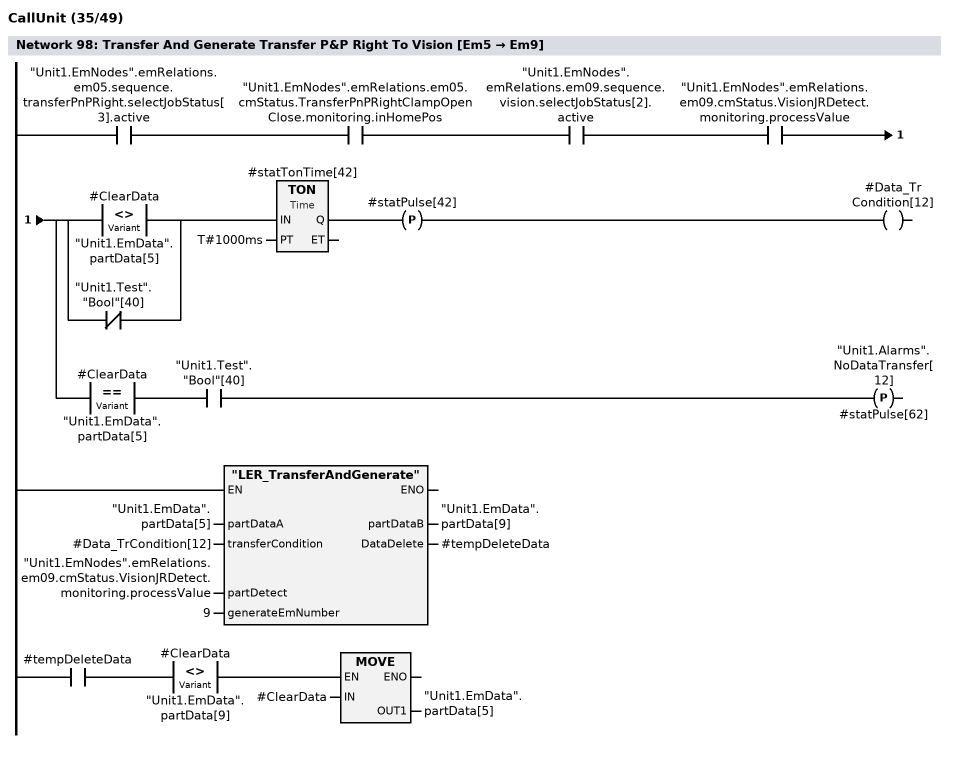
   #_w1 := "Unit1.EmNodes".emRelations.em05.sequence.transferPnPRight.selectJobStatus[3].active AND "Unit1.EmNodes".emRelations.em05.cmStatus.TransferPnPRightClampOpenClose.monitoring.inHomePos AND "Unit1.EmNodes".emRelations.em09.sequence.vision.selectJobStatus[2].active AND "Unit1.EmNodes".emRelations.em09.cmStatus.VisionJRDetect.monitoring.processValue;
   #statTonTime[42].TON(IN := #_w1 AND ((#ClearData <> "Unit1.EmData".partData[5]) OR NOT "Unit1.Test"."Bool"[40]),
                        PT := T#1000ms);
   #_w2 := #statTonTime[42].Q AND NOT #statPulse[42];   // rising edge
   #statPulse[42] := #statTonTime[42].Q;
   #Data_TrCondition[12] := #_w2;
   #_w3 := #_w1 AND (#ClearData = "Unit1.EmData".partData[5]) AND "Unit1.Test"."Bool"[40];
   "Unit1.Alarms".NoDataTransfer[12] := #_w3 AND NOT #statPulse[62];   // rising edge
   #statPulse[62] := #_w3;
   "LER_TransferAndGenerate"(partDataA := "Unit1.EmData".partData[5],
                           transferCondition := #Data_TrCondition[12],
                           partDetect := "Unit1.EmNodes".emRelations.em09.cmStatus.VisionJRDetect.monitoring.processValue,
                           generateEmNumber := 9,
                           partDataB => "Unit1.EmData".partData[9],
                           DataDelete => #tempDeleteData);
   IF #tempDeleteData AND (#ClearData <> "Unit1.EmData".partData[9]) THEN
       "Unit1.EmData".partData[5] := #ClearData;
   END_IF;
END_REGION

REGION Network 99: Transfer And Generate Vision To Transfer P&P Right [Em9 → Em5]
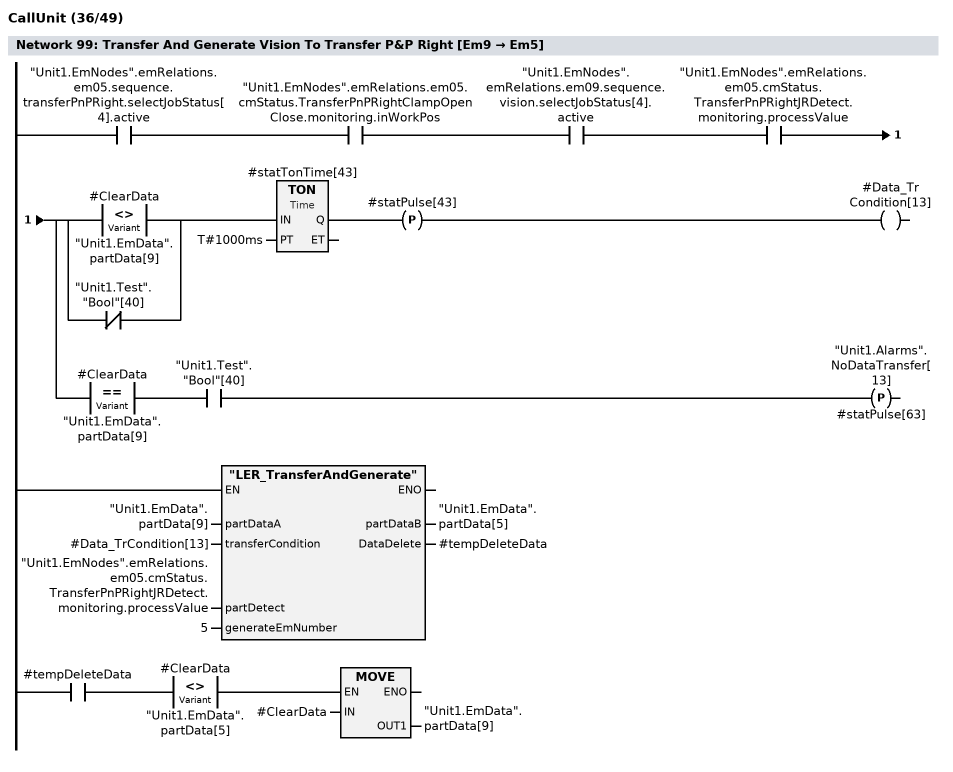
   #_w1 := "Unit1.EmNodes".emRelations.em05.sequence.transferPnPRight.selectJobStatus[4].active AND "Unit1.EmNodes".emRelations.em05.cmStatus.TransferPnPRightClampOpenClose.monitoring.inWorkPos AND "Unit1.EmNodes".emRelations.em09.sequence.vision.selectJobStatus[4].active AND "Unit1.EmNodes".emRelations.em05.cmStatus.TransferPnPRightJRDetect.monitoring.processValue;
   #statTonTime[43].TON(IN := #_w1 AND ((#ClearData <> "Unit1.EmData".partData[9]) OR NOT "Unit1.Test"."Bool"[40]),
                        PT := T#1000ms);
   #_w2 := #statTonTime[43].Q AND NOT #statPulse[43];   // rising edge
   #statPulse[43] := #statTonTime[43].Q;
   #Data_TrCondition[13] := #_w2;
   #_w3 := #_w1 AND (#ClearData = "Unit1.EmData".partData[9]) AND "Unit1.Test"."Bool"[40];
   "Unit1.Alarms".NoDataTransfer[13] := #_w3 AND NOT #statPulse[63];   // rising edge
   #statPulse[63] := #_w3;
   "LER_TransferAndGenerate"(partDataA := "Unit1.EmData".partData[9],
                           transferCondition := #Data_TrCondition[13],
                           partDetect := "Unit1.EmNodes".emRelations.em05.cmStatus.TransferPnPRightJRDetect.monitoring.processValue,
                           generateEmNumber := 5,
                           partDataB => "Unit1.EmData".partData[5],
                           DataDelete => #tempDeleteData);
   IF #tempDeleteData AND (#ClearData <> "Unit1.EmData".partData[5]) THEN
       "Unit1.EmData".partData[9] := #ClearData;
   END_IF;
END_REGION

REGION Network 100: Transfer And Generate Transfer P&P Right To Laser Mark [Em5 → Em10]
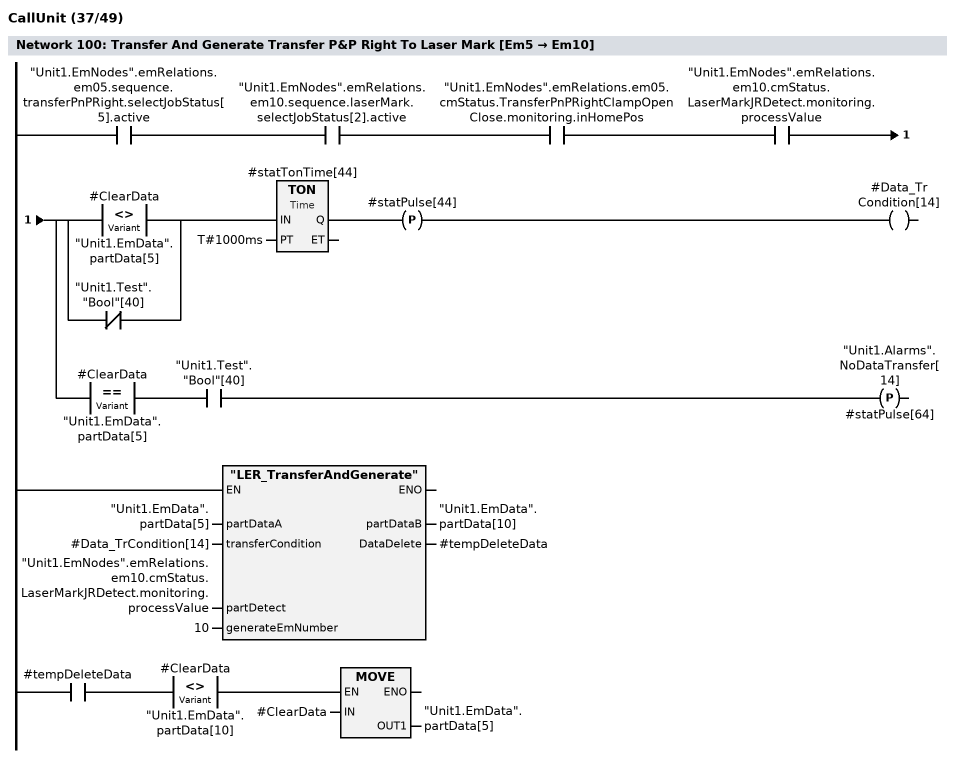
   #_w1 := "Unit1.EmNodes".emRelations.em05.sequence.transferPnPRight.selectJobStatus[5].active AND "Unit1.EmNodes".emRelations.em10.sequence.laserMark.selectJobStatus[2].active AND "Unit1.EmNodes".emRelations.em05.cmStatus.TransferPnPRightClampOpenClose.monitoring.inHomePos AND "Unit1.EmNodes".emRelations.em10.cmStatus.LaserMarkJRDetect.monitoring.processValue;
   #statTonTime[44].TON(IN := #_w1 AND ((#ClearData <> "Unit1.EmData".partData[5]) OR NOT "Unit1.Test"."Bool"[40]),
                        PT := T#1000ms);
   #_w2 := #statTonTime[44].Q AND NOT #statPulse[44];   // rising edge
   #statPulse[44] := #statTonTime[44].Q;
   #Data_TrCondition[14] := #_w2;
   #_w3 := #_w1 AND (#ClearData = "Unit1.EmData".partData[5]) AND "Unit1.Test"."Bool"[40];
   "Unit1.Alarms".NoDataTransfer[14] := #_w3 AND NOT #statPulse[64];   // rising edge
   #statPulse[64] := #_w3;
   "LER_TransferAndGenerate"(partDataA := "Unit1.EmData".partData[5],
                           transferCondition := #Data_TrCondition[14],
                           partDetect := "Unit1.EmNodes".emRelations.em10.cmStatus.LaserMarkJRDetect.monitoring.processValue,
                           generateEmNumber := 10,
                           partDataB => "Unit1.EmData".partData[10],
                           DataDelete => #tempDeleteData);
   IF #tempDeleteData AND (#ClearData <> "Unit1.EmData".partData[10]) THEN
       "Unit1.EmData".partData[5] := #ClearData;
   END_IF;
END_REGION

REGION Network 101: Transfer And Generate Laser Mark To Transfer P&P Right [Em10 → Em5]
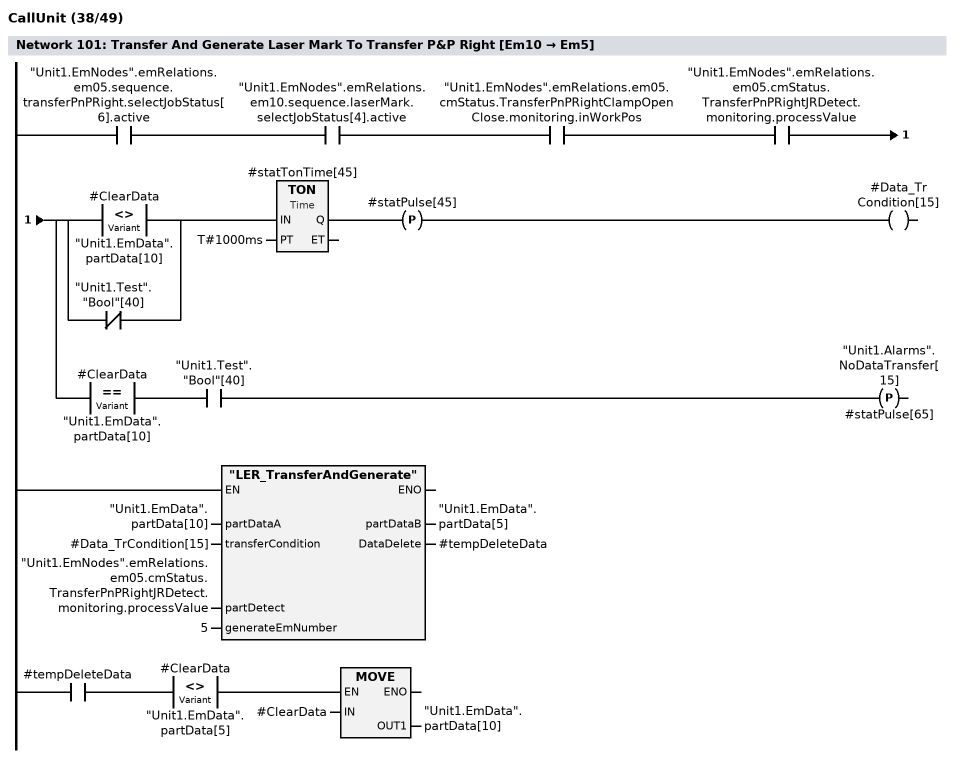
   #_w1 := "Unit1.EmNodes".emRelations.em05.sequence.transferPnPRight.selectJobStatus[6].active AND "Unit1.EmNodes".emRelations.em10.sequence.laserMark.selectJobStatus[4].active AND "Unit1.EmNodes".emRelations.em05.cmStatus.TransferPnPRightClampOpenClose.monitoring.inWorkPos AND "Unit1.EmNodes".emRelations.em05.cmStatus.TransferPnPRightJRDetect.monitoring.processValue;
   #statTonTime[45].TON(IN := #_w1 AND ((#ClearData <> "Unit1.EmData".partData[10]) OR NOT "Unit1.Test"."Bool"[40]),
                        PT := T#1000ms);
   #_w2 := #statTonTime[45].Q AND NOT #statPulse[45];   // rising edge
   #statPulse[45] := #statTonTime[45].Q;
   #Data_TrCondition[15] := #_w2;
   #_w3 := #_w1 AND (#ClearData = "Unit1.EmData".partData[10]) AND "Unit1.Test"."Bool"[40];
   "Unit1.Alarms".NoDataTransfer[15] := #_w3 AND NOT #statPulse[65];   // rising edge
   #statPulse[65] := #_w3;
   "LER_TransferAndGenerate"(partDataA := "Unit1.EmData".partData[10],
                           transferCondition := #Data_TrCondition[15],
                           partDetect := "Unit1.EmNodes".emRelations.em05.cmStatus.TransferPnPRightJRDetect.monitoring.processValue,
                           generateEmNumber := 5,
                           partDataB => "Unit1.EmData".partData[5],
                           DataDelete => #tempDeleteData);
   IF #tempDeleteData AND (#ClearData <> "Unit1.EmData".partData[5]) THEN
       "Unit1.EmData".partData[10] := #ClearData;
   END_IF;
END_REGION

REGION Network 102: Transfer And Generate Transfer P&P Right To Weight Check [Em5 → Em11]
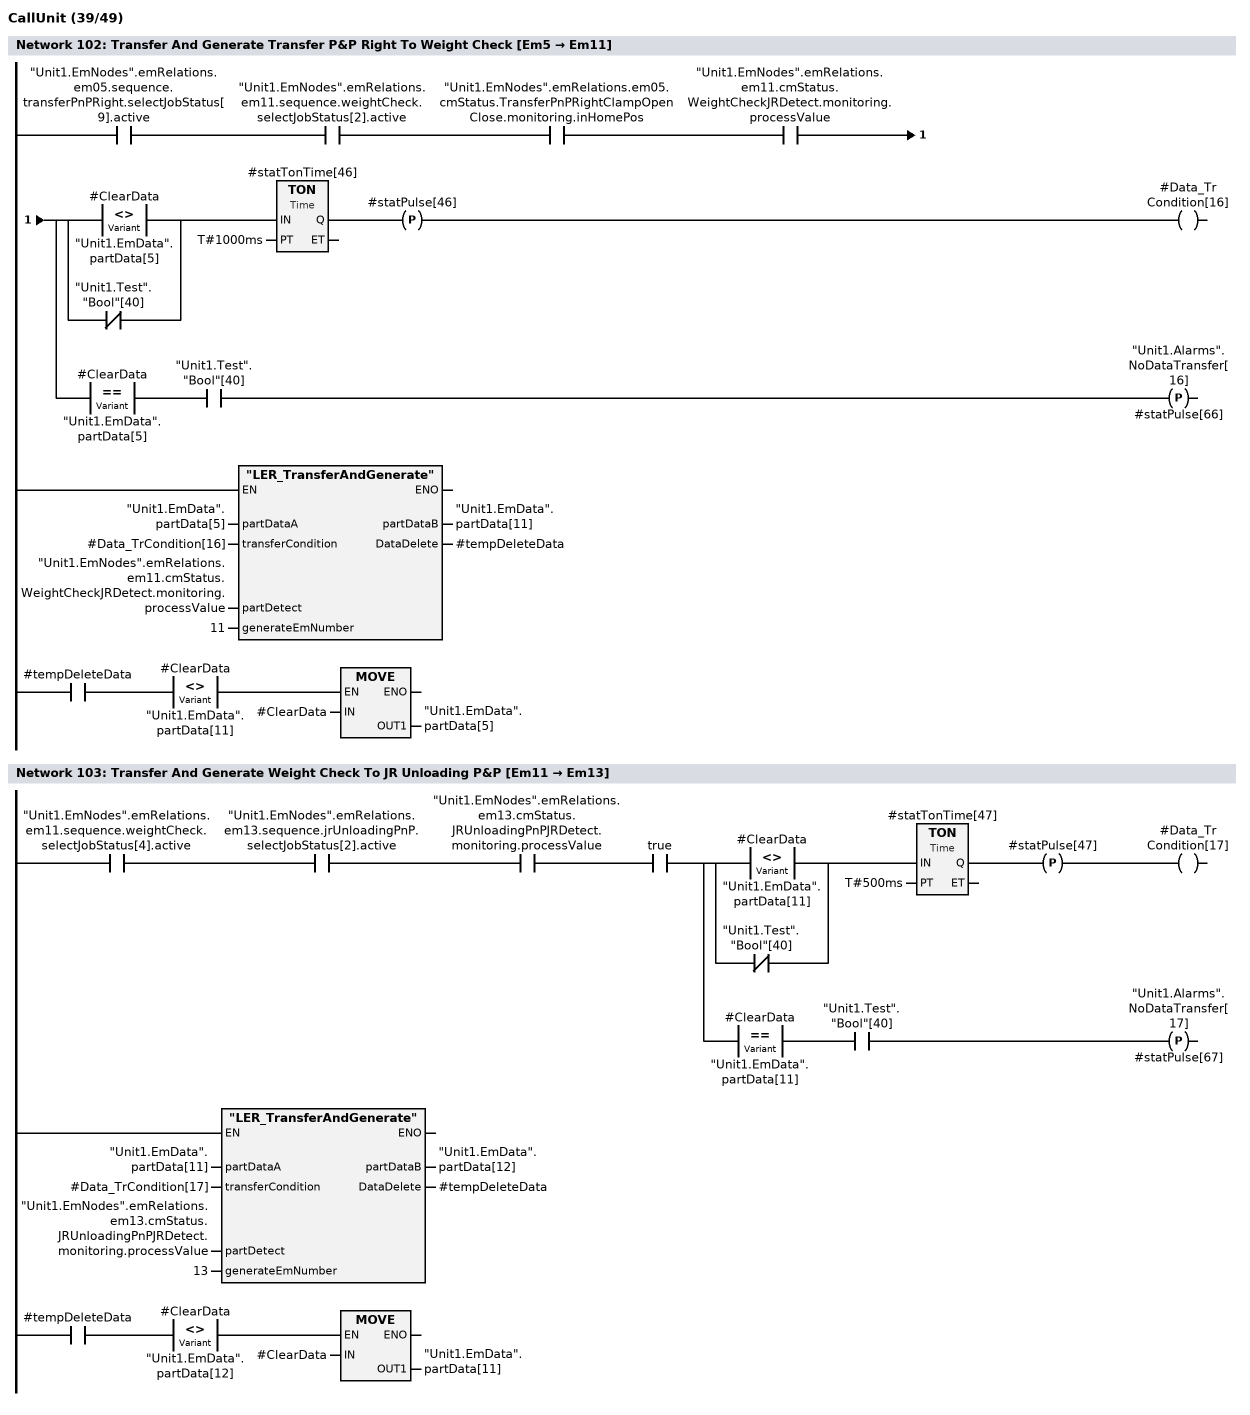
   #_w1 := "Unit1.EmNodes".emRelations.em05.sequence.transferPnPRight.selectJobStatus[9].active AND "Unit1.EmNodes".emRelations.em11.sequence.weightCheck.selectJobStatus[2].active AND "Unit1.EmNodes".emRelations.em05.cmStatus.TransferPnPRightClampOpenClose.monitoring.inHomePos AND "Unit1.EmNodes".emRelations.em11.cmStatus.WeightCheckJRDetect.monitoring.processValue;
   #statTonTime[46].TON(IN := #_w1 AND ((#ClearData <> "Unit1.EmData".partData[5]) OR NOT "Unit1.Test"."Bool"[40]),
                        PT := T#1000ms);
   #_w2 := #statTonTime[46].Q AND NOT #statPulse[46];   // rising edge
   #statPulse[46] := #statTonTime[46].Q;
   #Data_TrCondition[16] := #_w2;
   #_w3 := #_w1 AND (#ClearData = "Unit1.EmData".partData[5]) AND "Unit1.Test"."Bool"[40];
   "Unit1.Alarms".NoDataTransfer[16] := #_w3 AND NOT #statPulse[66];   // rising edge
   #statPulse[66] := #_w3;
   "LER_TransferAndGenerate"(partDataA := "Unit1.EmData".partData[5],
                           transferCondition := #Data_TrCondition[16],
                           partDetect := "Unit1.EmNodes".emRelations.em11.cmStatus.WeightCheckJRDetect.monitoring.processValue,
                           generateEmNumber := 11,
                           partDataB => "Unit1.EmData".partData[11],
                           DataDelete => #tempDeleteData);
   IF #tempDeleteData AND (#ClearData <> "Unit1.EmData".partData[11]) THEN
       "Unit1.EmData".partData[5] := #ClearData;
   END_IF;
END_REGION

REGION Network 103: Transfer And Generate Weight Check To JR Unloading P&P [Em11 → Em13]
   #_w1 := "Unit1.EmNodes".emRelations.em11.sequence.weightCheck.selectJobStatus[4].active AND "Unit1.EmNodes".emRelations.em13.sequence.jrUnloadingPnP.selectJobStatus[2].active AND "Unit1.EmNodes".emRelations.em13.cmStatus.JRUnloadingPnPJRDetect.monitoring.processValue AND true;
   #statTonTime[47].TON(IN := #_w1 AND ((#ClearData <> "Unit1.EmData".partData[11]) OR NOT "Unit1.Test"."Bool"[40]),
                        PT := T#500ms);
   #_w2 := #statTonTime[47].Q AND NOT #statPulse[47];   // rising edge
   #statPulse[47] := #statTonTime[47].Q;
   #Data_TrCondition[17] := #_w2;
   #_w3 := #_w1 AND (#ClearData = "Unit1.EmData".partData[11]) AND "Unit1.Test"."Bool"[40];
   "Unit1.Alarms".NoDataTransfer[17] := #_w3 AND NOT #statPulse[67];   // rising edge
   #statPulse[67] := #_w3;
   "LER_TransferAndGenerate"(partDataA := "Unit1.EmData".partData[11],
                           transferCondition := #Data_TrCondition[17],
                           partDetect := "Unit1.EmNodes".emRelations.em13.cmStatus.JRUnloadingPnPJRDetect.monitoring.processValue,
                           generateEmNumber := 13,
                           partDataB => "Unit1.EmData".partData[12],
                           DataDelete => #tempDeleteData);
   IF #tempDeleteData AND (#ClearData <> "Unit1.EmData".partData[12]) THEN
       "Unit1.EmData".partData[11] := #ClearData;
   END_IF;
END_REGION

REGION Network 104: Transfer And Generate JR Unloading P&P To ConveyorA [Em13 → ConveyorA]
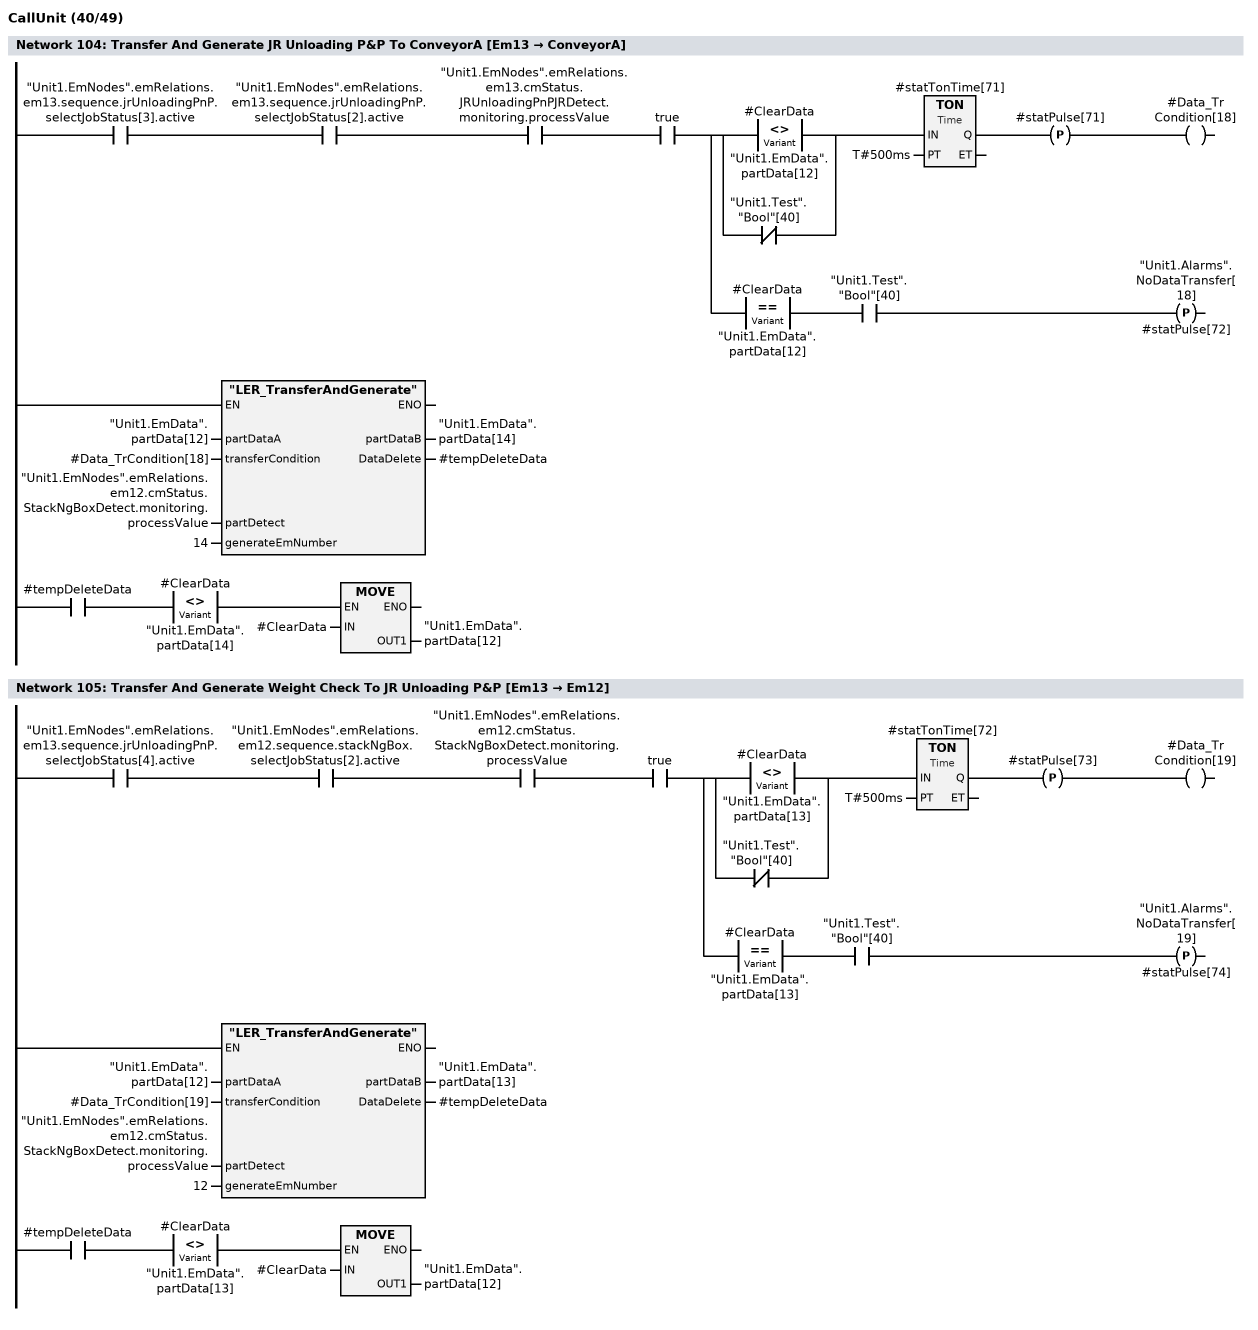
   #_w1 := "Unit1.EmNodes".emRelations.em13.sequence.jrUnloadingPnP.selectJobStatus[3].active AND "Unit1.EmNodes".emRelations.em13.sequence.jrUnloadingPnP.selectJobStatus[2].active AND "Unit1.EmNodes".emRelations.em13.cmStatus.JRUnloadingPnPJRDetect.monitoring.processValue AND true;
   #statTonTime[71].TON(IN := #_w1 AND ((#ClearData <> "Unit1.EmData".partData[12]) OR NOT "Unit1.Test"."Bool"[40]),
                        PT := T#500ms);
   #_w2 := #statTonTime[71].Q AND NOT #statPulse[71];   // rising edge
   #statPulse[71] := #statTonTime[71].Q;
   #Data_TrCondition[18] := #_w2;
   #_w3 := #_w1 AND (#ClearData = "Unit1.EmData".partData[12]) AND "Unit1.Test"."Bool"[40];
   "Unit1.Alarms".NoDataTransfer[18] := #_w3 AND NOT #statPulse[72];   // rising edge
   #statPulse[72] := #_w3;
   "LER_TransferAndGenerate"(partDataA := "Unit1.EmData".partData[12],
                           transferCondition := #Data_TrCondition[18],
                           partDetect := "Unit1.EmNodes".emRelations.em12.cmStatus.StackNgBoxDetect.monitoring.processValue,
                           generateEmNumber := 14,
                           partDataB => "Unit1.EmData".partData[14],
                           DataDelete => #tempDeleteData);
   IF #tempDeleteData AND (#ClearData <> "Unit1.EmData".partData[14]) THEN
       "Unit1.EmData".partData[12] := #ClearData;
   END_IF;
END_REGION

REGION Network 105: Transfer And Generate Weight Check To JR Unloading P&P [Em13 → Em12]
   #_w1 := "Unit1.EmNodes".emRelations.em13.sequence.jrUnloadingPnP.selectJobStatus[4].active AND "Unit1.EmNodes".emRelations.em12.sequence.stackNgBox.selectJobStatus[2].active AND "Unit1.EmNodes".emRelations.em12.cmStatus.StackNgBoxDetect.monitoring.processValue AND true;
   #statTonTime[72].TON(IN := #_w1 AND ((#ClearData <> "Unit1.EmData".partData[13]) OR NOT "Unit1.Test"."Bool"[40]),
                        PT := T#500ms);
   #_w2 := #statTonTime[72].Q AND NOT #statPulse[73];   // rising edge
   #statPulse[73] := #statTonTime[72].Q;
   #Data_TrCondition[19] := #_w2;
   #_w3 := #_w1 AND (#ClearData = "Unit1.EmData".partData[13]) AND "Unit1.Test"."Bool"[40];
   "Unit1.Alarms".NoDataTransfer[19] := #_w3 AND NOT #statPulse[74];   // rising edge
   #statPulse[74] := #_w3;
   "LER_TransferAndGenerate"(partDataA := "Unit1.EmData".partData[12],
                           transferCondition := #Data_TrCondition[19],
                           partDetect := "Unit1.EmNodes".emRelations.em12.cmStatus.StackNgBoxDetect.monitoring.processValue,
                           generateEmNumber := 12,
                           partDataB => "Unit1.EmData".partData[13],
                           DataDelete => #tempDeleteData);
   IF #tempDeleteData AND (#ClearData <> "Unit1.EmData".partData[13]) THEN
       "Unit1.EmData".partData[12] := #ClearData;
   END_IF;
END_REGION

REGION Network 106: Data Delete
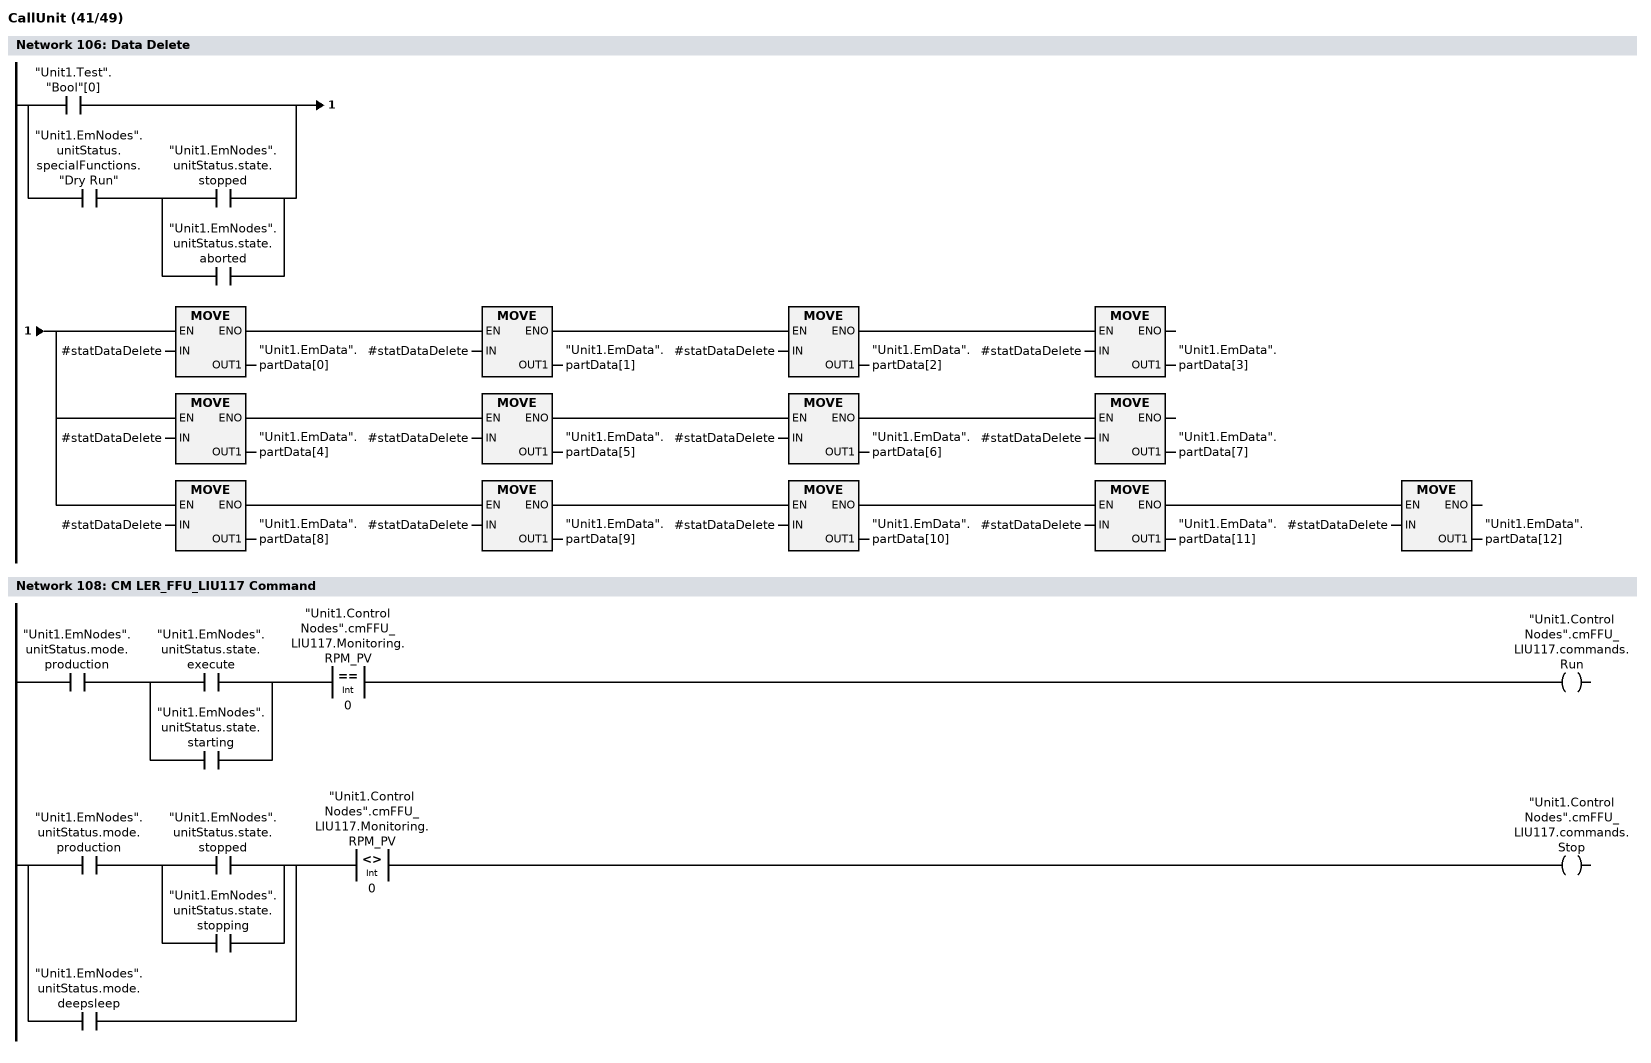
   RUNG wire#powerrail
      Contact( "Unit1.Test"."Bool"[0] )
      wire#w1
      Move(in := #statDataDelete, out1 => "Unit1.EmData".partData[0])
      Move(in := #statDataDelete, out1 => "Unit1.EmData".partData[1])
      Move(in := #statDataDelete, out1 => "Unit1.EmData".partData[2])
      Move(in := #statDataDelete, out1 => "Unit1.EmData".partData[3])
   END_RUNG
   RUNG wire#powerrail
      Contact( "Unit1.EmNodes".unitStatus.specialFunctions."Dry Run" )
      wire#w2
      Contact( "Unit1.EmNodes".unitStatus.state.stopped )
   END_RUNG wire#w1
   RUNG wire#w2
      Contact( "Unit1.EmNodes".unitStatus.state.aborted )
   END_RUNG wire#w1
   RUNG wire#w1
      Move(in := #statDataDelete, out1 => "Unit1.EmData".partData[4])
      Move(in := #statDataDelete, out1 => "Unit1.EmData".partData[5])
      Move(in := #statDataDelete, out1 => "Unit1.EmData".partData[6])
      Move(in := #statDataDelete, out1 => "Unit1.EmData".partData[7])
   END_RUNG
   RUNG wire#w1
      Move(in := #statDataDelete, out1 => "Unit1.EmData".partData[8])
      Move(in := #statDataDelete, out1 => "Unit1.EmData".partData[9])
      Move(in := #statDataDelete, out1 => "Unit1.EmData".partData[10])
      Move(in := #statDataDelete, out1 => "Unit1.EmData".partData[11])
      Move(in := #statDataDelete, out1 => "Unit1.EmData".partData[12])
   END_RUNG
   // the same network as SCL:
   IF "Unit1.Test"."Bool"[0] OR ("Unit1.EmNodes".unitStatus.specialFunctions."Dry Run" AND ("Unit1.EmNodes".unitStatus.state.stopped OR "Unit1.EmNodes".unitStatus.state.aborted)) THEN
       "Unit1.EmData".partData[0] := #statDataDelete;
       "Unit1.EmData".partData[1] := #statDataDelete;
       "Unit1.EmData".partData[2] := #statDataDelete;
       "Unit1.EmData".partData[3] := #statDataDelete;
       "Unit1.EmData".partData[4] := #statDataDelete;
       "Unit1.EmData".partData[5] := #statDataDelete;
       "Unit1.EmData".partData[6] := #statDataDelete;
       "Unit1.EmData".partData[7] := #statDataDelete;
       "Unit1.EmData".partData[8] := #statDataDelete;
       "Unit1.EmData".partData[9] := #statDataDelete;
       "Unit1.EmData".partData[10] := #statDataDelete;
       "Unit1.EmData".partData[11] := #statDataDelete;
       "Unit1.EmData".partData[12] := #statDataDelete;
   END_IF;
END_REGION

REGION Network 107: ******************** FFU LIU117 (MCU) ********************
END_REGION

REGION Network 108: CM LER_FFU_LIU117 Command
   RUNG wire#powerrail
      Contact( "Unit1.EmNodes".unitStatus.mode.production )
      wire#w1
      Contact( "Unit1.EmNodes".unitStatus.state.execute )
      wire#w2
      { S7_Templates := "SrcType := Int" } EQ_Contact(in1 := "Unit1.ControlNodes".cmFFU_LIU117.Monitoring.RPM_PV, in2 := 0)
      Coil( "Unit1.ControlNodes".cmFFU_LIU117.commands.Run )
   END_RUNG
   RUNG wire#w1
      Contact( "Unit1.EmNodes".unitStatus.state.starting )
   END_RUNG wire#w2
   RUNG wire#powerrail
      Contact( "Unit1.EmNodes".unitStatus.mode.production )
      wire#w3
      Contact( "Unit1.EmNodes".unitStatus.state.stopped )
      wire#w4
      { S7_Templates := "SrcType := Int" } NE_Contact(in1 := "Unit1.ControlNodes".cmFFU_LIU117.Monitoring.RPM_PV, in2 := 0)
      Coil( "Unit1.ControlNodes".cmFFU_LIU117.commands.Stop )
   END_RUNG
   RUNG wire#w3
      Contact( "Unit1.EmNodes".unitStatus.state.stopping )
   END_RUNG wire#w4
   RUNG wire#powerrail
      Contact( "Unit1.EmNodes".unitStatus.mode.deepsleep )
   END_RUNG wire#w4
   // the same network as SCL:
   "Unit1.ControlNodes".cmFFU_LIU117.commands.Run := "Unit1.EmNodes".unitStatus.mode.production AND ("Unit1.EmNodes".unitStatus.state.execute OR "Unit1.EmNodes".unitStatus.state.starting) AND ("Unit1.ControlNodes".cmFFU_LIU117.Monitoring.RPM_PV = 0);
   "Unit1.ControlNodes".cmFFU_LIU117.commands.Stop := (("Unit1.EmNodes".unitStatus.mode.production AND ("Unit1.EmNodes".unitStatus.state.stopped OR "Unit1.EmNodes".unitStatus.state.stopping)) OR "Unit1.EmNodes".unitStatus.mode.deepsleep) AND ("Unit1.ControlNodes".cmFFU_LIU117.Monitoring.RPM_PV <> 0);
END_REGION

REGION Network 109: Call LER_FFU_LU117
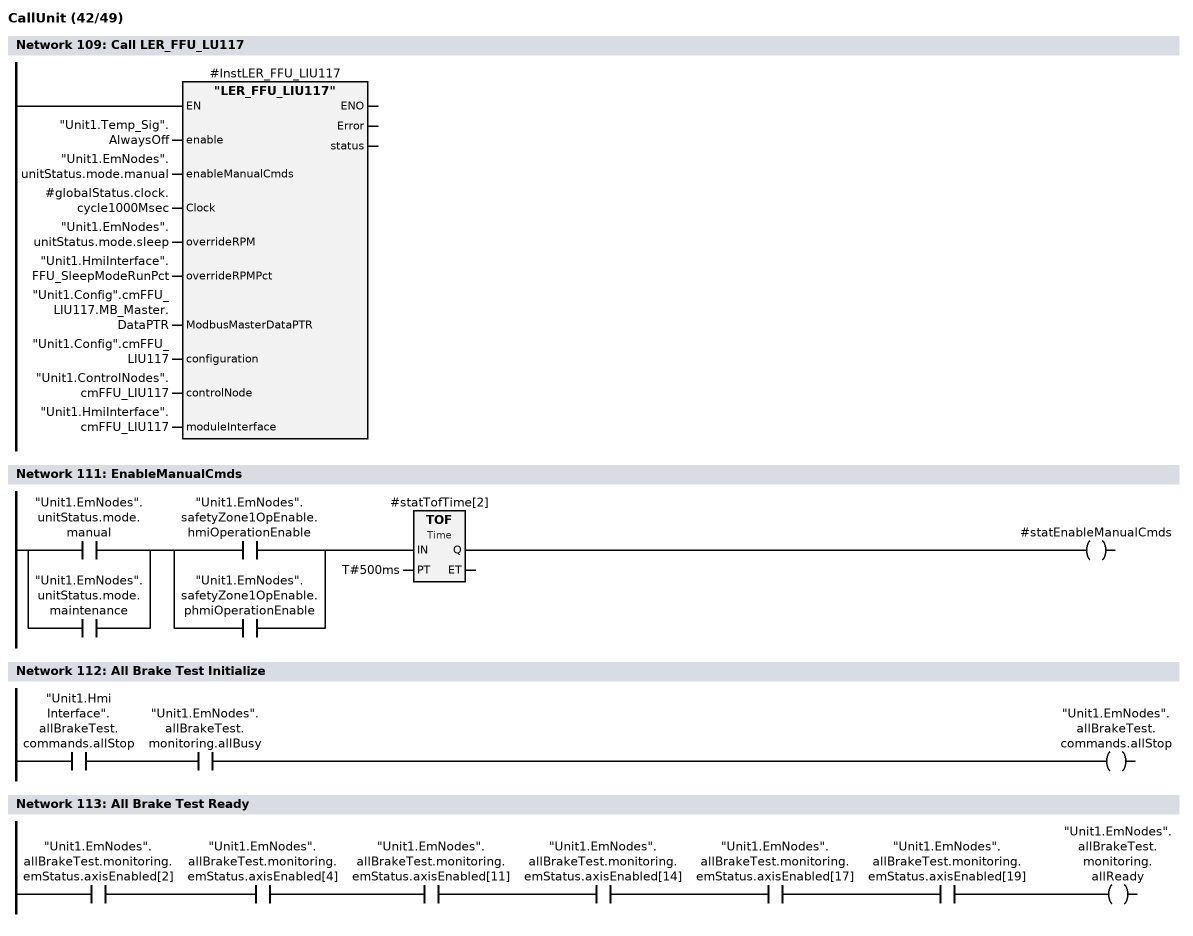
   RUNG wire#powerrail
      #InstLER_FFU_LIU117(enable := "Unit1.Temp_Sig".AlwaysOff, enableManualCmds := "Unit1.EmNodes".unitStatus.mode.manual, Clock := #globalStatus.clock.cycle1000Msec, overrideRPM := "Unit1.EmNodes".unitStatus.mode.sleep, overrideRPMPct := "Unit1.HmiInterface".FFU_SleepModeRunPct, ModbusMasterDataPTR := "Unit1.Config".cmFFU_LIU117.MB_Master.DataPTR, configuration := "Unit1.Config".cmFFU_LIU117, controlNode := "Unit1.ControlNodes".cmFFU_LIU117, moduleInterface := "Unit1.HmiInterface".cmFFU_LIU117, Error =>, status =>)
   END_RUNG
   // the same network as SCL:
   #InstLER_FFU_LIU117(enable := "Unit1.Temp_Sig".AlwaysOff,   // "LER_FFU_LIU117"
                       enableManualCmds := "Unit1.EmNodes".unitStatus.mode.manual,
                       Clock := #globalStatus.clock.cycle1000Msec,
                       overrideRPM := "Unit1.EmNodes".unitStatus.mode.sleep,
                       overrideRPMPct := "Unit1.HmiInterface".FFU_SleepModeRunPct,
                       ModbusMasterDataPTR := "Unit1.Config".cmFFU_LIU117.MB_Master.DataPTR,
                       configuration := "Unit1.Config".cmFFU_LIU117,
                       controlNode := "Unit1.ControlNodes".cmFFU_LIU117,
                       moduleInterface := "Unit1.HmiInterface".cmFFU_LIU117);
END_REGION

REGION Network 110: ******************** Brake Test ********************
END_REGION

REGION Network 111: EnableManualCmds
   RUNG wire#powerrail
      Contact( "Unit1.EmNodes".unitStatus.mode.manual )
      wire#w1
      Contact( "Unit1.EmNodes".safetyZone1OpEnable.hmiOperationEnable )
      wire#w2
      { S7_Templates := "time_type := Time" } #statTofTime[2].TOF(pt := T#500ms, et =>)
      Coil( #statEnableManualCmds )
   END_RUNG
   RUNG wire#powerrail
      Contact( "Unit1.EmNodes".unitStatus.mode.maintenance )
   END_RUNG wire#w1
   RUNG wire#w1
      Contact( "Unit1.EmNodes".safetyZone1OpEnable.phmiOperationEnable )
   END_RUNG wire#w2
   // the same network as SCL:
   #statTofTime[2].TOF(IN := ("Unit1.EmNodes".unitStatus.mode.manual OR "Unit1.EmNodes".unitStatus.mode.maintenance) AND ("Unit1.EmNodes".safetyZone1OpEnable.hmiOperationEnable OR "Unit1.EmNodes".safetyZone1OpEnable.phmiOperationEnable),
                       PT := T#500ms);
   #statEnableManualCmds := #statTofTime[2].Q;
END_REGION

REGION Network 112: All Brake Test Initialize
   RUNG wire#powerrail
      Contact( "Unit1.HmiInterface".allBrakeTest.commands.allStop )
      Contact( "Unit1.EmNodes".allBrakeTest.monitoring.allBusy )
      Coil( "Unit1.EmNodes".allBrakeTest.commands.allStop )
   END_RUNG
   // the same network as SCL:
   "Unit1.EmNodes".allBrakeTest.commands.allStop := "Unit1.HmiInterface".allBrakeTest.commands.allStop AND "Unit1.EmNodes".allBrakeTest.monitoring.allBusy;
END_REGION

REGION Network 113: All Brake Test Ready
   RUNG wire#powerrail
      Contact( "Unit1.EmNodes".allBrakeTest.monitoring.emStatus.axisEnabled[2] )
      Contact( "Unit1.EmNodes".allBrakeTest.monitoring.emStatus.axisEnabled[4] )
      Contact( "Unit1.EmNodes".allBrakeTest.monitoring.emStatus.axisEnabled[11] )
      Contact( "Unit1.EmNodes".allBrakeTest.monitoring.emStatus.axisEnabled[14] )
      Contact( "Unit1.EmNodes".allBrakeTest.monitoring.emStatus.axisEnabled[17] )
      Contact( "Unit1.EmNodes".allBrakeTest.monitoring.emStatus.axisEnabled[19] )
      Coil( "Unit1.EmNodes".allBrakeTest.monitoring.allReady )
   END_RUNG
   // the same network as SCL:
   "Unit1.EmNodes".allBrakeTest.monitoring.allReady := "Unit1.EmNodes".allBrakeTest.monitoring.emStatus.axisEnabled[2] AND "Unit1.EmNodes".allBrakeTest.monitoring.emStatus.axisEnabled[4] AND "Unit1.EmNodes".allBrakeTest.monitoring.emStatus.axisEnabled[11] AND "Unit1.EmNodes".allBrakeTest.monitoring.emStatus.axisEnabled[14] AND "Unit1.EmNodes".allBrakeTest.monitoring.emStatus.axisEnabled[17] AND "Unit1.EmNodes".allBrakeTest.monitoring.emStatus.axisEnabled[19];
END_REGION

REGION Network 114: All Brake Test Commands
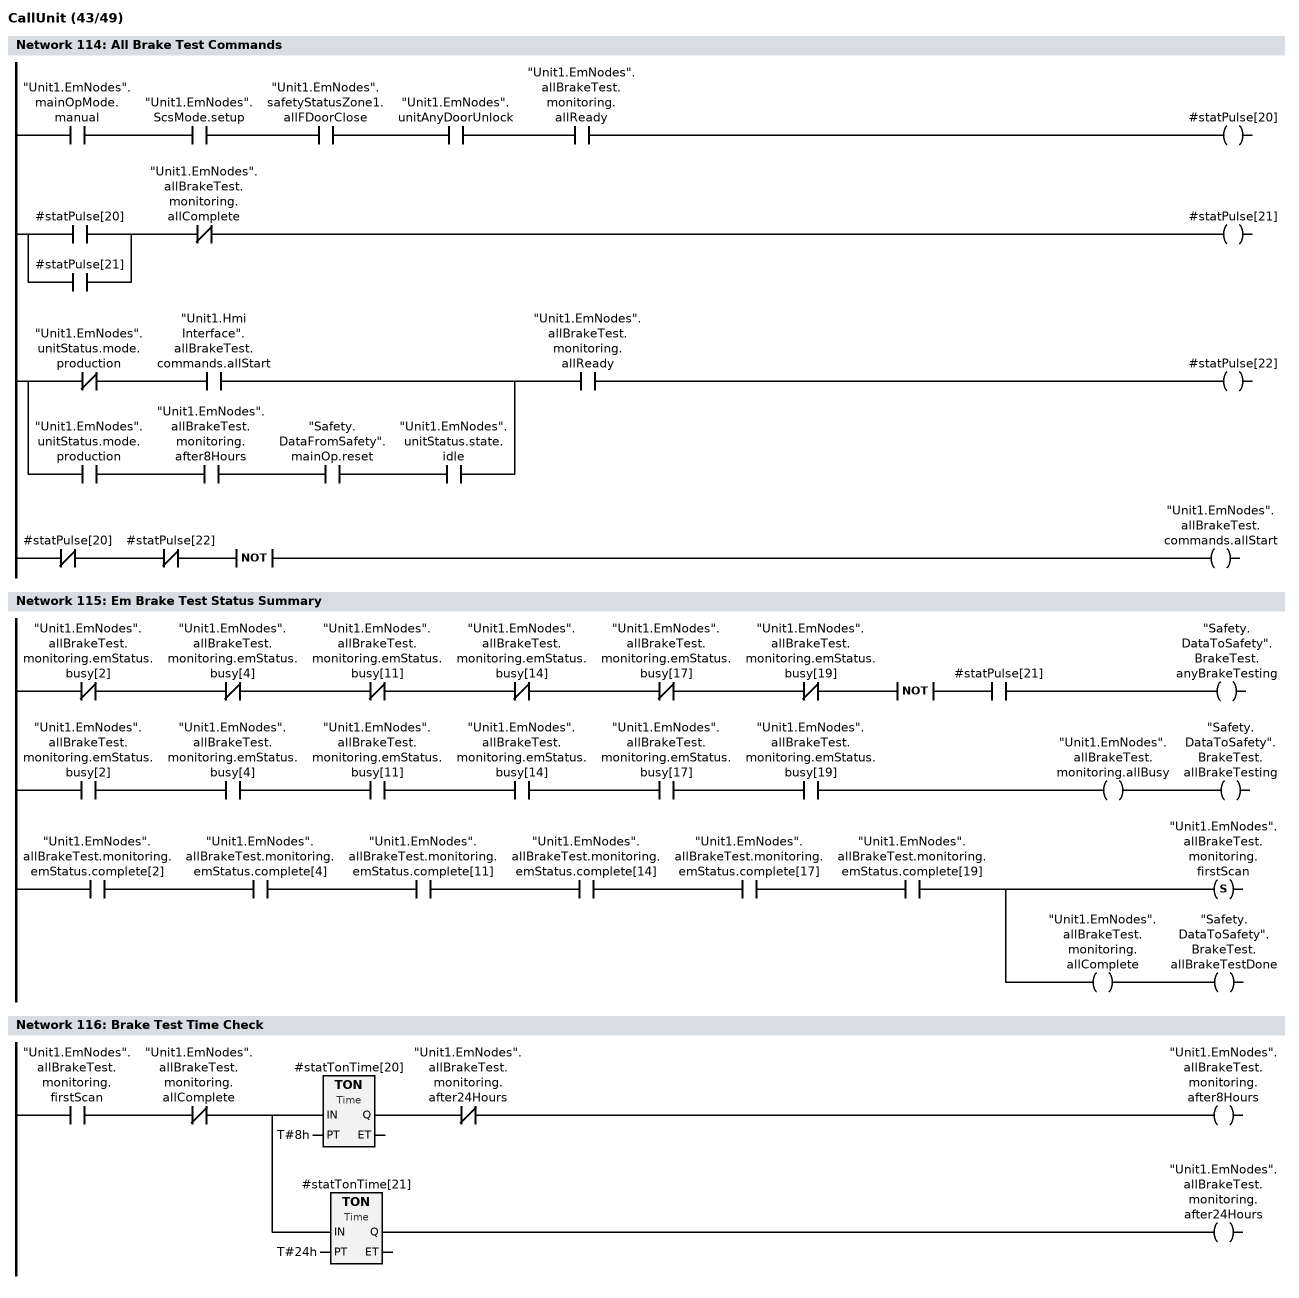
   RUNG wire#powerrail
      Contact( "Unit1.EmNodes".mainOpMode.manual )
      Contact( "Unit1.EmNodes".ScsMode.setup )
      Contact( "Unit1.EmNodes".safetyStatusZone1.allFDoorClose )
      Contact( "Unit1.EmNodes".unitAnyDoorUnlock )
      Contact( "Unit1.EmNodes".allBrakeTest.monitoring.allReady )
      Coil( #statPulse[20] )
   END_RUNG
   RUNG wire#powerrail
      Contact( #statPulse[20] )
      wire#w1
      I_Contact( "Unit1.EmNodes".allBrakeTest.monitoring.allComplete )
      Coil( #statPulse[21] )
   END_RUNG
   RUNG wire#powerrail
      Contact( #statPulse[21] )
   END_RUNG wire#w1
   RUNG wire#powerrail
      I_Contact( "Unit1.EmNodes".unitStatus.mode.production )
      Contact( "Unit1.HmiInterface".allBrakeTest.commands.allStart )
      wire#w2
      Contact( "Unit1.EmNodes".allBrakeTest.monitoring.allReady )
      Coil( #statPulse[22] )
   END_RUNG
   RUNG wire#powerrail
      Contact( "Unit1.EmNodes".unitStatus.mode.production )
      Contact( "Unit1.EmNodes".allBrakeTest.monitoring.after8Hours )
      Contact( "Safety.DataFromSafety".mainOp.reset )
      Contact( "Unit1.EmNodes".unitStatus.state.idle )
   END_RUNG wire#w2
   RUNG wire#powerrail
      I_Contact( #statPulse[20] )
      I_Contact( #statPulse[22] )
      Not()
      Coil( "Unit1.EmNodes".allBrakeTest.commands.allStart )
   END_RUNG
   // the same network as SCL:
   #statPulse[20] := "Unit1.EmNodes".mainOpMode.manual AND "Unit1.EmNodes".ScsMode.setup AND "Unit1.EmNodes".safetyStatusZone1.allFDoorClose AND "Unit1.EmNodes".unitAnyDoorUnlock AND "Unit1.EmNodes".allBrakeTest.monitoring.allReady;
   #statPulse[21] := (#statPulse[20] OR #statPulse[21]) AND NOT "Unit1.EmNodes".allBrakeTest.monitoring.allComplete;
   #statPulse[22] := ((NOT "Unit1.EmNodes".unitStatus.mode.production AND "Unit1.HmiInterface".allBrakeTest.commands.allStart) OR ("Unit1.EmNodes".unitStatus.mode.production AND "Unit1.EmNodes".allBrakeTest.monitoring.after8Hours AND "Safety.DataFromSafety".mainOp.reset AND "Unit1.EmNodes".unitStatus.state.idle)) AND "Unit1.EmNodes".allBrakeTest.monitoring.allReady;
   "Unit1.EmNodes".allBrakeTest.commands.allStart := NOT (NOT #statPulse[20] AND NOT #statPulse[22]);
END_REGION

REGION Network 115: Em Brake Test Status Summary
   RUNG wire#powerrail
      I_Contact( "Unit1.EmNodes".allBrakeTest.monitoring.emStatus.busy[2] )
      I_Contact( "Unit1.EmNodes".allBrakeTest.monitoring.emStatus.busy[4] )
      I_Contact( "Unit1.EmNodes".allBrakeTest.monitoring.emStatus.busy[11] )
      I_Contact( "Unit1.EmNodes".allBrakeTest.monitoring.emStatus.busy[14] )
      I_Contact( "Unit1.EmNodes".allBrakeTest.monitoring.emStatus.busy[17] )
      I_Contact( "Unit1.EmNodes".allBrakeTest.monitoring.emStatus.busy[19] )
      Not()
      Contact( #statPulse[21] )
      Coil( "Safety.DataToSafety".BrakeTest.anyBrakeTesting )
   END_RUNG
   RUNG wire#powerrail
      Contact( "Unit1.EmNodes".allBrakeTest.monitoring.emStatus.busy[2] )
      Contact( "Unit1.EmNodes".allBrakeTest.monitoring.emStatus.busy[4] )
      Contact( "Unit1.EmNodes".allBrakeTest.monitoring.emStatus.busy[11] )
      Contact( "Unit1.EmNodes".allBrakeTest.monitoring.emStatus.busy[14] )
      Contact( "Unit1.EmNodes".allBrakeTest.monitoring.emStatus.busy[17] )
      Contact( "Unit1.EmNodes".allBrakeTest.monitoring.emStatus.busy[19] )
      Coil( "Unit1.EmNodes".allBrakeTest.monitoring.allBusy )
      Coil( "Safety.DataToSafety".BrakeTest.allBrakeTesting )
   END_RUNG
   RUNG wire#powerrail
      Contact( "Unit1.EmNodes".allBrakeTest.monitoring.emStatus.complete[2] )
      Contact( "Unit1.EmNodes".allBrakeTest.monitoring.emStatus.complete[4] )
      Contact( "Unit1.EmNodes".allBrakeTest.monitoring.emStatus.complete[11] )
      Contact( "Unit1.EmNodes".allBrakeTest.monitoring.emStatus.complete[14] )
      Contact( "Unit1.EmNodes".allBrakeTest.monitoring.emStatus.complete[17] )
      Contact( "Unit1.EmNodes".allBrakeTest.monitoring.emStatus.complete[19] )
      wire#w1
      S_Coil( "Unit1.EmNodes".allBrakeTest.monitoring.firstScan )
   END_RUNG
   RUNG wire#w1
      Coil( "Unit1.EmNodes".allBrakeTest.monitoring.allComplete )
      Coil( "Safety.DataToSafety".BrakeTest.allBrakeTestDone )
   END_RUNG
   // the same network as SCL:
   "Safety.DataToSafety".BrakeTest.anyBrakeTesting := NOT (NOT "Unit1.EmNodes".allBrakeTest.monitoring.emStatus.busy[2] AND NOT "Unit1.EmNodes".allBrakeTest.monitoring.emStatus.busy[4] AND NOT "Unit1.EmNodes".allBrakeTest.monitoring.emStatus.busy[11] AND NOT "Unit1.EmNodes".allBrakeTest.monitoring.emStatus.busy[14] AND NOT "Unit1.EmNodes".allBrakeTest.monitoring.emStatus.busy[17] AND NOT "Unit1.EmNodes".allBrakeTest.monitoring.emStatus.busy[19]) AND #statPulse[21];
   "Unit1.EmNodes".allBrakeTest.monitoring.allBusy := "Unit1.EmNodes".allBrakeTest.monitoring.emStatus.busy[2] AND "Unit1.EmNodes".allBrakeTest.monitoring.emStatus.busy[4] AND "Unit1.EmNodes".allBrakeTest.monitoring.emStatus.busy[11] AND "Unit1.EmNodes".allBrakeTest.monitoring.emStatus.busy[14] AND "Unit1.EmNodes".allBrakeTest.monitoring.emStatus.busy[17] AND "Unit1.EmNodes".allBrakeTest.monitoring.emStatus.busy[19];
   "Safety.DataToSafety".BrakeTest.allBrakeTesting := "Unit1.EmNodes".allBrakeTest.monitoring.allBusy;
   #_w1 := "Unit1.EmNodes".allBrakeTest.monitoring.emStatus.complete[2] AND "Unit1.EmNodes".allBrakeTest.monitoring.emStatus.complete[4] AND "Unit1.EmNodes".allBrakeTest.monitoring.emStatus.complete[11] AND "Unit1.EmNodes".allBrakeTest.monitoring.emStatus.complete[14] AND "Unit1.EmNodes".allBrakeTest.monitoring.emStatus.complete[17] AND "Unit1.EmNodes".allBrakeTest.monitoring.emStatus.complete[19];
   IF #_w1 THEN "Unit1.EmNodes".allBrakeTest.monitoring.firstScan := TRUE; END_IF;
   "Unit1.EmNodes".allBrakeTest.monitoring.allComplete := #_w1;
   "Safety.DataToSafety".BrakeTest.allBrakeTestDone := #_w1;
END_REGION

REGION Network 116: Brake Test Time Check
   RUNG wire#powerrail
      Contact( "Unit1.EmNodes".allBrakeTest.monitoring.firstScan )
      I_Contact( "Unit1.EmNodes".allBrakeTest.monitoring.allComplete )
      wire#w1
      { S7_Templates := "time_type := Time" } #statTonTime[20].TON(pt := T#8h, et =>)
      I_Contact( "Unit1.EmNodes".allBrakeTest.monitoring.after24Hours )
      Coil( "Unit1.EmNodes".allBrakeTest.monitoring.after8Hours )
   END_RUNG
   RUNG wire#w1
      { S7_Templates := "time_type := Time" } #statTonTime[21].TON(pt := T#24h, et =>)
      Coil( "Unit1.EmNodes".allBrakeTest.monitoring.after24Hours )
   END_RUNG
   // the same network as SCL:
   #_w1 := "Unit1.EmNodes".allBrakeTest.monitoring.firstScan AND NOT "Unit1.EmNodes".allBrakeTest.monitoring.allComplete;
   #statTonTime[20].TON(IN := #_w1, PT := T#8h);
   "Unit1.EmNodes".allBrakeTest.monitoring.after8Hours := #statTonTime[20].Q AND NOT "Unit1.EmNodes".allBrakeTest.monitoring.after24Hours;
   #statTonTime[21].TON(IN := #_w1, PT := T#24h);
   "Unit1.EmNodes".allBrakeTest.monitoring.after24Hours := #statTonTime[21].Q;
END_REGION

REGION Network 117: All Brake Test Monitoring
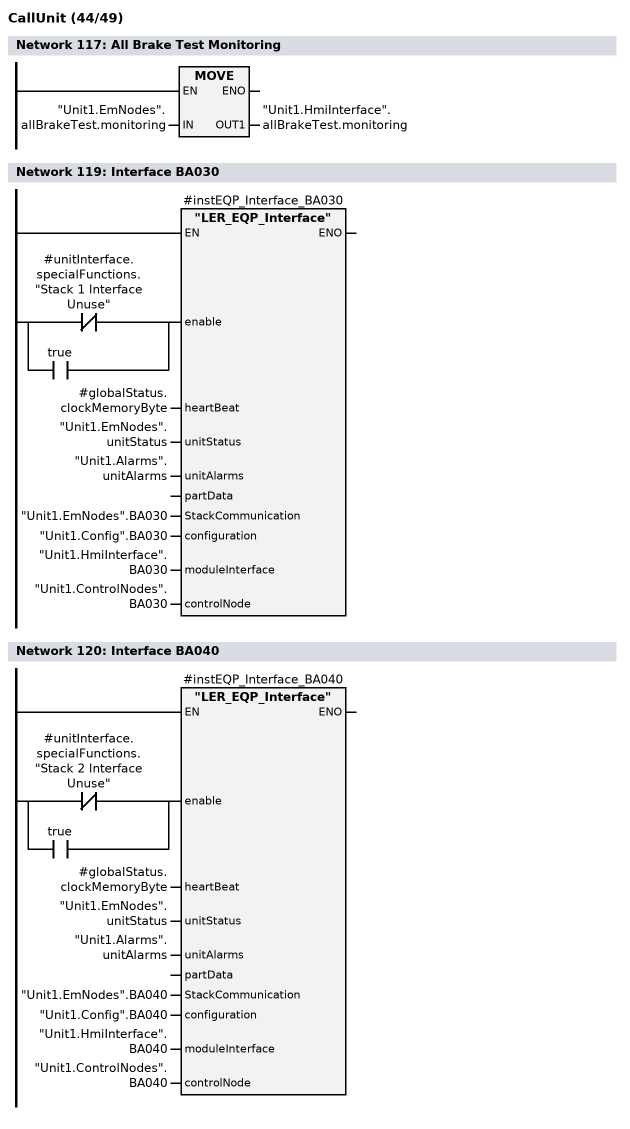
   RUNG wire#powerrail
      Move(in := "Unit1.EmNodes".allBrakeTest.monitoring, out1 => "Unit1.HmiInterface".allBrakeTest.monitoring)
   END_RUNG
   // the same network as SCL:
   "Unit1.HmiInterface".allBrakeTest.monitoring := "Unit1.EmNodes".allBrakeTest.monitoring;
END_REGION

REGION Network 118: ******************** PLC Communication ********************
END_REGION

REGION Network 119: Interface BA030
   RUNG wire#powerrail
      #instEQP_Interface_BA030(enable := wire#w1, heartBeat := #globalStatus.clockMemoryByte, unitStatus := "Unit1.EmNodes".unitStatus, unitAlarms := "Unit1.Alarms".unitAlarms, partData :=, StackCommunication := "Unit1.EmNodes".BA030, configuration := "Unit1.Config".BA030, moduleInterface := "Unit1.HmiInterface".BA030, controlNode := "Unit1.ControlNodes".BA030)
   END_RUNG
   RUNG wire#powerrail
      I_Contact( #unitInterface.specialFunctions."Stack 1 lnterface Unuse" )
   END_RUNG wire#w1
   RUNG wire#powerrail
      Contact( true )
   END_RUNG wire#w1
   // the same network as SCL:
   #instEQP_Interface_BA030(enable := NOT #unitInterface.specialFunctions."Stack 1 lnterface Unuse" OR true,   // "LER_EQP_Interface"
                           heartBeat := #globalStatus.clockMemoryByte,
                           unitStatus := "Unit1.EmNodes".unitStatus,
                           unitAlarms := "Unit1.Alarms".unitAlarms,
                           StackCommunication := "Unit1.EmNodes".BA030,
                           configuration := "Unit1.Config".BA030,
                           moduleInterface := "Unit1.HmiInterface".BA030,
                           controlNode := "Unit1.ControlNodes".BA030);
END_REGION

REGION Network 120: Interface BA040
   RUNG wire#powerrail
      #instEQP_Interface_BA040(enable := wire#w1, heartBeat := #globalStatus.clockMemoryByte, unitStatus := "Unit1.EmNodes".unitStatus, unitAlarms := "Unit1.Alarms".unitAlarms, partData :=, StackCommunication := "Unit1.EmNodes".BA040, configuration := "Unit1.Config".BA040, moduleInterface := "Unit1.HmiInterface".BA040, controlNode := "Unit1.ControlNodes".BA040)
   END_RUNG
   RUNG wire#powerrail
      I_Contact( #unitInterface.specialFunctions."Stack 2 lnterface Unuse" )
   END_RUNG wire#w1
   RUNG wire#powerrail
      Contact( true )
   END_RUNG wire#w1
   // the same network as SCL:
   #instEQP_Interface_BA040(enable := NOT #unitInterface.specialFunctions."Stack 2 lnterface Unuse" OR true,   // "LER_EQP_Interface"
                           heartBeat := #globalStatus.clockMemoryByte,
                           unitStatus := "Unit1.EmNodes".unitStatus,
                           unitAlarms := "Unit1.Alarms".unitAlarms,
                           StackCommunication := "Unit1.EmNodes".BA040,
                           configuration := "Unit1.Config".BA040,
                           moduleInterface := "Unit1.HmiInterface".BA040,
                           controlNode := "Unit1.ControlNodes".BA040);
END_REGION

REGION Network 121: Interface BA100
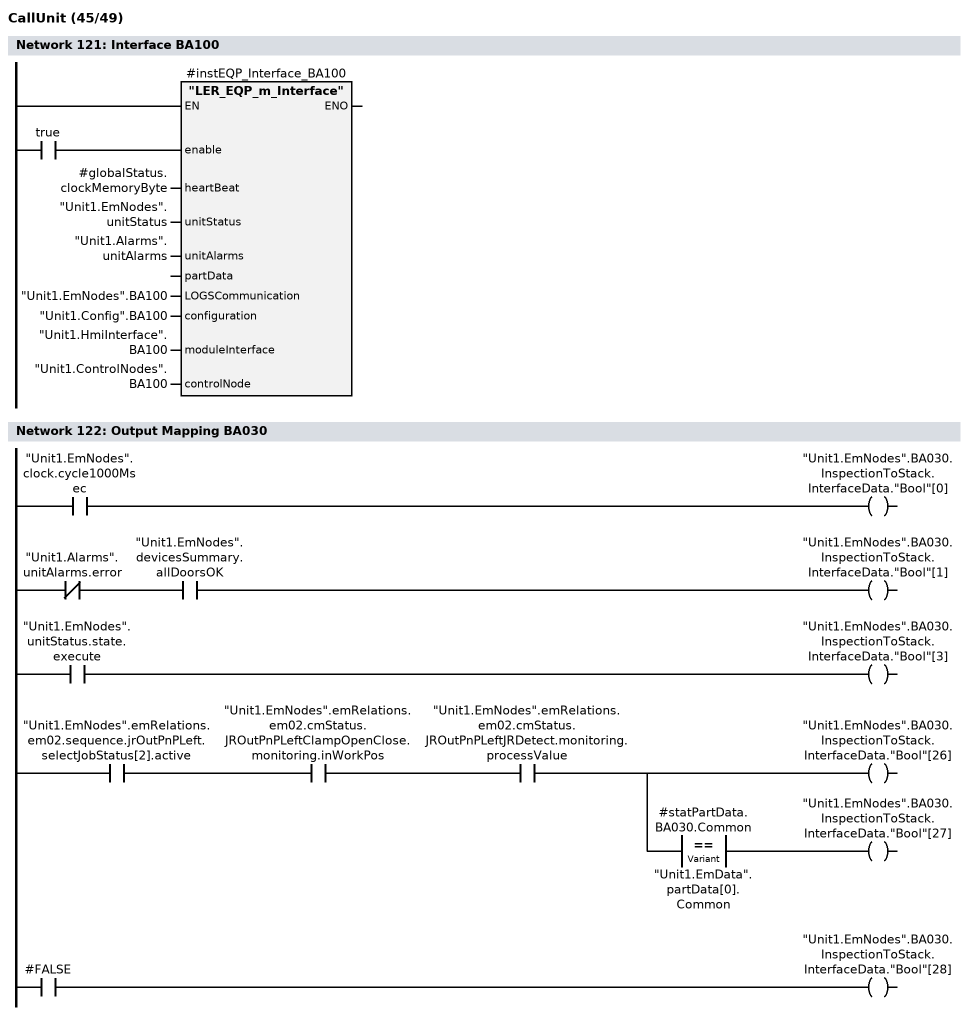
   RUNG wire#powerrail
      #instEQP_Interface_BA100(enable := wire#w1, heartBeat := #globalStatus.clockMemoryByte, unitStatus := "Unit1.EmNodes".unitStatus, unitAlarms := "Unit1.Alarms".unitAlarms, partData :=, LOGSCommunication := "Unit1.EmNodes".BA100, configuration := "Unit1.Config".BA100, moduleInterface := "Unit1.HmiInterface".BA100, controlNode := "Unit1.ControlNodes".BA100)
   END_RUNG
   RUNG wire#powerrail
      Contact( true )
   END_RUNG wire#w1
   // the same network as SCL:
   #instEQP_Interface_BA100(enable := true,   // "LER_EQP_m_Interface"
                           heartBeat := #globalStatus.clockMemoryByte,
                           unitStatus := "Unit1.EmNodes".unitStatus,
                           unitAlarms := "Unit1.Alarms".unitAlarms,
                           LOGSCommunication := "Unit1.EmNodes".BA100,
                           configuration := "Unit1.Config".BA100,
                           moduleInterface := "Unit1.HmiInterface".BA100,
                           controlNode := "Unit1.ControlNodes".BA100);
END_REGION

REGION Network 122: Output Mapping BA030
   RUNG wire#powerrail
      Contact( "Unit1.EmNodes".clock.cycle1000Msec )
      Coil( "Unit1.EmNodes".BA030.InspectionToStack.InterfaceData."Bool"[0] )
   END_RUNG
   RUNG wire#powerrail
      I_Contact( "Unit1.Alarms".unitAlarms.error )
      Contact( "Unit1.EmNodes".devicesSummary.allDoorsOK )
      Coil( "Unit1.EmNodes".BA030.InspectionToStack.InterfaceData."Bool"[1] )
   END_RUNG
   RUNG wire#powerrail
      Contact( "Unit1.EmNodes".unitStatus.state.execute )
      Coil( "Unit1.EmNodes".BA030.InspectionToStack.InterfaceData."Bool"[3] )
   END_RUNG
   RUNG wire#powerrail
      Contact( "Unit1.EmNodes".emRelations.em02.sequence.jrOutPnPLeft.selectJobStatus[2].active )
      Contact( "Unit1.EmNodes".emRelations.em02.cmStatus.JROutPnPLeftClampOpenClose.monitoring.inWorkPos )
      Contact( "Unit1.EmNodes".emRelations.em02.cmStatus.JROutPnPLeftJRDetect.monitoring.processValue )
      wire#w1
      Coil( "Unit1.EmNodes".BA030.InspectionToStack.InterfaceData."Bool"[26] )
   END_RUNG
   RUNG wire#w1
      { S7_Templates := "SrcType := Variant" } EQ_Contact(in1 := #statPartData.BA030.Common, in2 := "Unit1.EmData".partData[0].Common)
      Coil( "Unit1.EmNodes".BA030.InspectionToStack.InterfaceData."Bool"[27] )
   END_RUNG
   RUNG wire#powerrail
      Contact( #FALSE )
      Coil( "Unit1.EmNodes".BA030.InspectionToStack.InterfaceData."Bool"[28] )
   END_RUNG
   // the same network as SCL:
   "Unit1.EmNodes".BA030.InspectionToStack.InterfaceData."Bool"[0] := "Unit1.EmNodes".clock.cycle1000Msec;
   "Unit1.EmNodes".BA030.InspectionToStack.InterfaceData."Bool"[1] := NOT "Unit1.Alarms".unitAlarms.error AND "Unit1.EmNodes".devicesSummary.allDoorsOK;
   "Unit1.EmNodes".BA030.InspectionToStack.InterfaceData."Bool"[3] := "Unit1.EmNodes".unitStatus.state.execute;
   "Unit1.EmNodes".BA030.InspectionToStack.InterfaceData."Bool"[26] := "Unit1.EmNodes".emRelations.em02.sequence.jrOutPnPLeft.selectJobStatus[2].active AND "Unit1.EmNodes".emRelations.em02.cmStatus.JROutPnPLeftClampOpenClose.monitoring.inWorkPos AND "Unit1.EmNodes".emRelations.em02.cmStatus.JROutPnPLeftJRDetect.monitoring.processValue;
   "Unit1.EmNodes".BA030.InspectionToStack.InterfaceData."Bool"[27] := "Unit1.EmNodes".emRelations.em02.sequence.jrOutPnPLeft.selectJobStatus[2].active AND "Unit1.EmNodes".emRelations.em02.cmStatus.JROutPnPLeftClampOpenClose.monitoring.inWorkPos AND "Unit1.EmNodes".emRelations.em02.cmStatus.JROutPnPLeftJRDetect.monitoring.processValue AND (#statPartData.BA030.Common = "Unit1.EmData".partData[0].Common);
   "Unit1.EmNodes".BA030.InspectionToStack.InterfaceData."Bool"[28] := #FALSE;
END_REGION

REGION Network 123: Output Mapping BA040
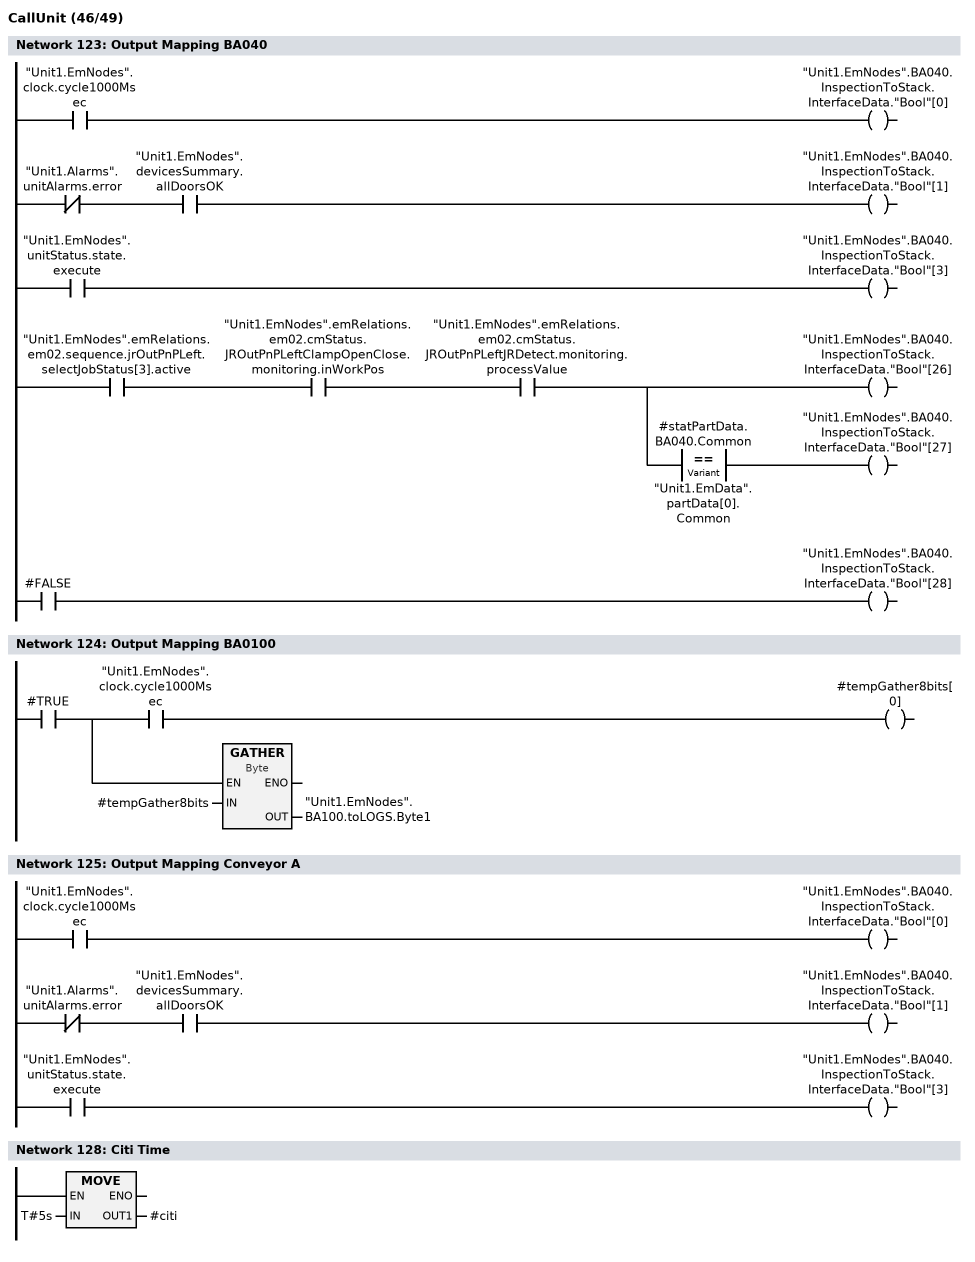
   RUNG wire#powerrail
      Contact( "Unit1.EmNodes".clock.cycle1000Msec )
      Coil( "Unit1.EmNodes".BA040.InspectionToStack.InterfaceData."Bool"[0] )
   END_RUNG
   RUNG wire#powerrail
      I_Contact( "Unit1.Alarms".unitAlarms.error )
      Contact( "Unit1.EmNodes".devicesSummary.allDoorsOK )
      Coil( "Unit1.EmNodes".BA040.InspectionToStack.InterfaceData."Bool"[1] )
   END_RUNG
   RUNG wire#powerrail
      Contact( "Unit1.EmNodes".unitStatus.state.execute )
      Coil( "Unit1.EmNodes".BA040.InspectionToStack.InterfaceData."Bool"[3] )
   END_RUNG
   RUNG wire#powerrail
      Contact( "Unit1.EmNodes".emRelations.em02.sequence.jrOutPnPLeft.selectJobStatus[3].active )
      Contact( "Unit1.EmNodes".emRelations.em02.cmStatus.JROutPnPLeftClampOpenClose.monitoring.inWorkPos )
      Contact( "Unit1.EmNodes".emRelations.em02.cmStatus.JROutPnPLeftJRDetect.monitoring.processValue )
      wire#w1
      Coil( "Unit1.EmNodes".BA040.InspectionToStack.InterfaceData."Bool"[26] )
   END_RUNG
   RUNG wire#w1
      { S7_Templates := "SrcType := Variant" } EQ_Contact(in1 := #statPartData.BA040.Common, in2 := "Unit1.EmData".partData[0].Common)
      Coil( "Unit1.EmNodes".BA040.InspectionToStack.InterfaceData."Bool"[27] )
   END_RUNG
   RUNG wire#powerrail
      Contact( #FALSE )
      Coil( "Unit1.EmNodes".BA040.InspectionToStack.InterfaceData."Bool"[28] )
   END_RUNG
   // the same network as SCL:
   "Unit1.EmNodes".BA040.InspectionToStack.InterfaceData."Bool"[0] := "Unit1.EmNodes".clock.cycle1000Msec;
   "Unit1.EmNodes".BA040.InspectionToStack.InterfaceData."Bool"[1] := NOT "Unit1.Alarms".unitAlarms.error AND "Unit1.EmNodes".devicesSummary.allDoorsOK;
   "Unit1.EmNodes".BA040.InspectionToStack.InterfaceData."Bool"[3] := "Unit1.EmNodes".unitStatus.state.execute;
   "Unit1.EmNodes".BA040.InspectionToStack.InterfaceData."Bool"[26] := "Unit1.EmNodes".emRelations.em02.sequence.jrOutPnPLeft.selectJobStatus[3].active AND "Unit1.EmNodes".emRelations.em02.cmStatus.JROutPnPLeftClampOpenClose.monitoring.inWorkPos AND "Unit1.EmNodes".emRelations.em02.cmStatus.JROutPnPLeftJRDetect.monitoring.processValue;
   "Unit1.EmNodes".BA040.InspectionToStack.InterfaceData."Bool"[27] := "Unit1.EmNodes".emRelations.em02.sequence.jrOutPnPLeft.selectJobStatus[3].active AND "Unit1.EmNodes".emRelations.em02.cmStatus.JROutPnPLeftClampOpenClose.monitoring.inWorkPos AND "Unit1.EmNodes".emRelations.em02.cmStatus.JROutPnPLeftJRDetect.monitoring.processValue AND (#statPartData.BA040.Common = "Unit1.EmData".partData[0].Common);
   "Unit1.EmNodes".BA040.InspectionToStack.InterfaceData."Bool"[28] := #FALSE;
END_REGION

REGION Network 124: Output Mapping BA0100
   RUNG wire#powerrail
      Contact( #TRUE )
      wire#w1
      Contact( "Unit1.EmNodes".clock.cycle1000Msec )
      Coil( #tempGather8bits[0] )
   END_RUNG
   RUNG wire#w1
      { S7_Templates := "[dest_type := Byte, src_type := Bool]" } GATHER(IN := #tempGather8bits, OUT => "Unit1.EmNodes".BA100.toLOGS.Byte1)
   END_RUNG
   // the same network as SCL:
   #tempGather8bits[0] := #TRUE AND "Unit1.EmNodes".clock.cycle1000Msec;
   IF #TRUE THEN GATHER(IN := #tempGather8bits, OUT => "Unit1.EmNodes".BA100.toLOGS.Byte1); END_IF;
END_REGION

REGION Network 125: Output Mapping Conveyor A
   RUNG wire#powerrail
      Contact( "Unit1.EmNodes".clock.cycle1000Msec )
      Coil( "Unit1.EmNodes".BA040.InspectionToStack.InterfaceData."Bool"[0] )
   END_RUNG
   RUNG wire#powerrail
      I_Contact( "Unit1.Alarms".unitAlarms.error )
      Contact( "Unit1.EmNodes".devicesSummary.allDoorsOK )
      Coil( "Unit1.EmNodes".BA040.InspectionToStack.InterfaceData."Bool"[1] )
   END_RUNG
   RUNG wire#powerrail
      Contact( "Unit1.EmNodes".unitStatus.state.execute )
      Coil( "Unit1.EmNodes".BA040.InspectionToStack.InterfaceData."Bool"[3] )
   END_RUNG
   // the same network as SCL:
   "Unit1.EmNodes".BA040.InspectionToStack.InterfaceData."Bool"[0] := "Unit1.EmNodes".clock.cycle1000Msec;
   "Unit1.EmNodes".BA040.InspectionToStack.InterfaceData."Bool"[1] := NOT "Unit1.Alarms".unitAlarms.error AND "Unit1.EmNodes".devicesSummary.allDoorsOK;
   "Unit1.EmNodes".BA040.InspectionToStack.InterfaceData."Bool"[3] := "Unit1.EmNodes".unitStatus.state.execute;
END_REGION

REGION Network 127: ******************** CITI ********************
END_REGION

REGION Network 128: Citi Time
   RUNG wire#powerrail
      Move(in := T#5s, out1 => #citi)
   END_RUNG
   // the same network as SCL:
   #citi := T#5s;
END_REGION

REGION Network 129: Auto Cycle Running 0
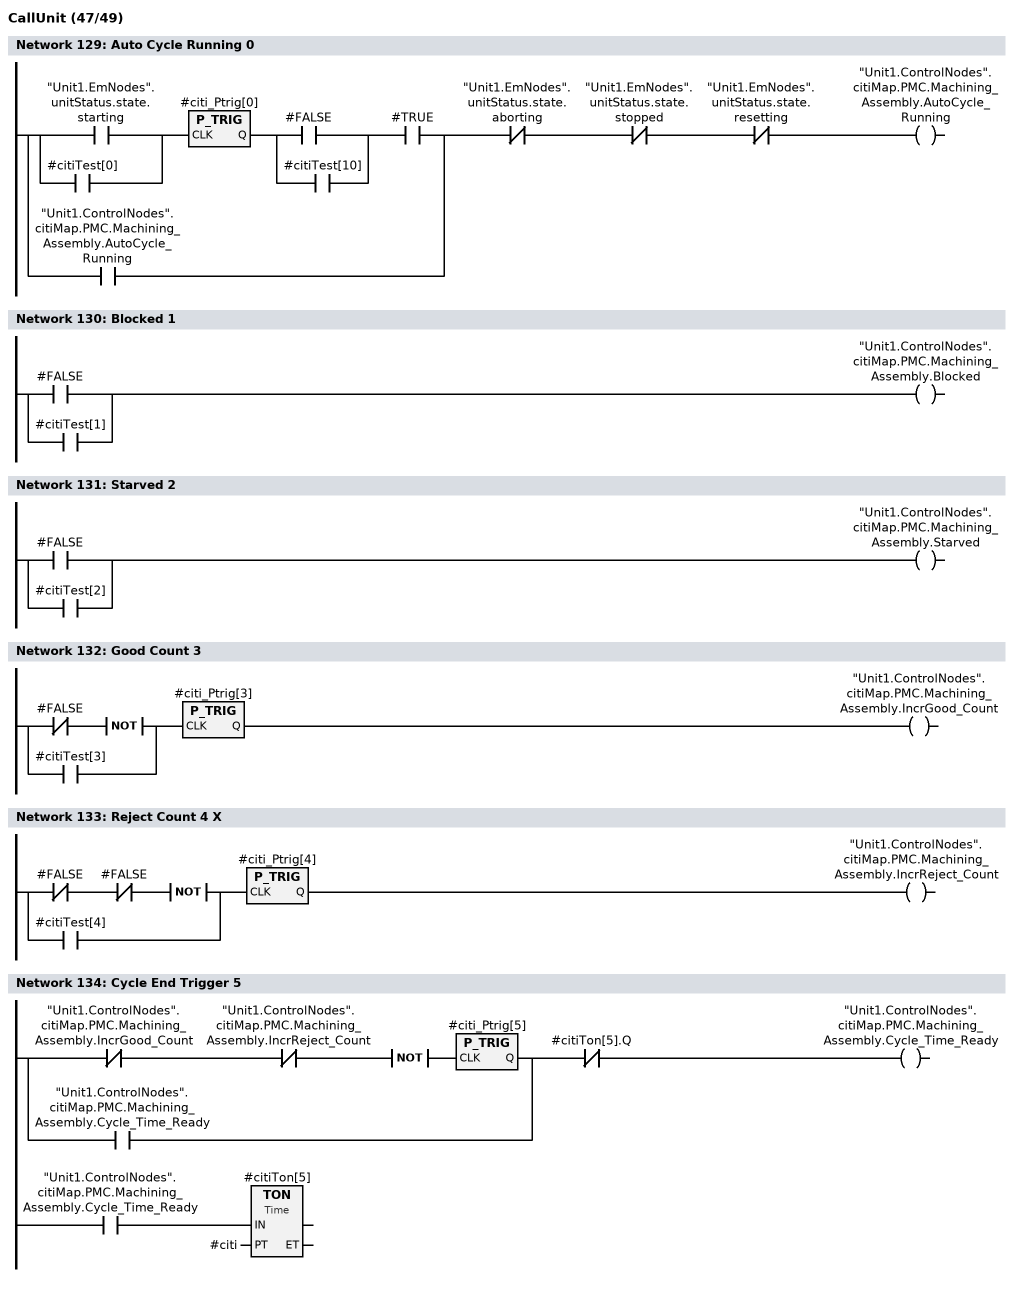
   RUNG wire#powerrail
      Contact( "Unit1.EmNodes".unitStatus.state.starting )
      wire#w1
      P_Trig( #citi_Ptrig[0] )
      wire#w2
      Contact( #FALSE )
      wire#w3
      Contact( #TRUE )
      wire#w4
      I_Contact( "Unit1.EmNodes".unitStatus.state.aborting )
      I_Contact( "Unit1.EmNodes".unitStatus.state.stopped )
      I_Contact( "Unit1.EmNodes".unitStatus.state.resetting )
      Coil( "Unit1.ControlNodes".citiMap.PMC.Machining_Assembly.AutoCycle_Running )
   END_RUNG
   RUNG wire#powerrail
      Contact( #citiTest[0] )
   END_RUNG wire#w1
   RUNG wire#w2
      Contact( #citiTest[10] )
   END_RUNG wire#w3
   RUNG wire#powerrail
      Contact( "Unit1.ControlNodes".citiMap.PMC.Machining_Assembly.AutoCycle_Running )
   END_RUNG wire#w4
   // the same network as SCL:
   #_w1 := "Unit1.EmNodes".unitStatus.state.starting OR #citiTest[0];
   #_w2 := #_w1 AND NOT #citi_Ptrig[0];   // rising edge
   #citi_Ptrig[0] := #_w1;
   "Unit1.ControlNodes".citiMap.PMC.Machining_Assembly.AutoCycle_Running := ((#_w2 AND (#FALSE OR #citiTest[10]) AND #TRUE) OR "Unit1.ControlNodes".citiMap.PMC.Machining_Assembly.AutoCycle_Running) AND NOT "Unit1.EmNodes".unitStatus.state.aborting AND NOT "Unit1.EmNodes".unitStatus.state.stopped AND NOT "Unit1.EmNodes".unitStatus.state.resetting;
END_REGION

REGION Network 130: Blocked 1
   RUNG wire#powerrail
      Contact( #FALSE )
      wire#w1
      Coil( "Unit1.ControlNodes".citiMap.PMC.Machining_Assembly.Blocked )
   END_RUNG
   RUNG wire#powerrail
      Contact( #citiTest[1] )
   END_RUNG wire#w1
   // the same network as SCL:
   "Unit1.ControlNodes".citiMap.PMC.Machining_Assembly.Blocked := #FALSE OR #citiTest[1];
END_REGION

REGION Network 131: Starved 2
   RUNG wire#powerrail
      Contact( #FALSE )
      wire#w1
      Coil( "Unit1.ControlNodes".citiMap.PMC.Machining_Assembly.Starved )
   END_RUNG
   RUNG wire#powerrail
      Contact( #citiTest[2] )
   END_RUNG wire#w1
   // the same network as SCL:
   "Unit1.ControlNodes".citiMap.PMC.Machining_Assembly.Starved := #FALSE OR #citiTest[2];
END_REGION

REGION Network 132: Good Count 3
   RUNG wire#powerrail
      I_Contact( #FALSE )
      Not()
      wire#w1
      P_Trig( #citi_Ptrig[3] )
      Coil( "Unit1.ControlNodes".citiMap.PMC.Machining_Assembly.IncrGood_Count )
   END_RUNG
   RUNG wire#powerrail
      Contact( #citiTest[3] )
   END_RUNG wire#w1
   // the same network as SCL:
   #_w1 := NOT (NOT #FALSE) OR #citiTest[3];
   #_w2 := #_w1 AND NOT #citi_Ptrig[3];   // rising edge
   #citi_Ptrig[3] := #_w1;
   "Unit1.ControlNodes".citiMap.PMC.Machining_Assembly.IncrGood_Count := #_w2;
END_REGION

REGION Network 133: Reject Count 4 X
   RUNG wire#powerrail
      I_Contact( #FALSE )
      I_Contact( #FALSE )
      Not()
      wire#w1
      P_Trig( #citi_Ptrig[4] )
      Coil( "Unit1.ControlNodes".citiMap.PMC.Machining_Assembly.IncrReject_Count )
   END_RUNG
   RUNG wire#powerrail
      Contact( #citiTest[4] )
   END_RUNG wire#w1
   // the same network as SCL:
   #_w1 := NOT (NOT #FALSE AND NOT #FALSE) OR #citiTest[4];
   #_w2 := #_w1 AND NOT #citi_Ptrig[4];   // rising edge
   #citi_Ptrig[4] := #_w1;
   "Unit1.ControlNodes".citiMap.PMC.Machining_Assembly.IncrReject_Count := #_w2;
END_REGION

REGION Network 134: Cycle End Trigger 5
   RUNG wire#powerrail
      I_Contact( "Unit1.ControlNodes".citiMap.PMC.Machining_Assembly.IncrGood_Count )
      I_Contact( "Unit1.ControlNodes".citiMap.PMC.Machining_Assembly.IncrReject_Count )
      Not()
      P_Trig( #citi_Ptrig[5] )
      wire#w1
      I_Contact( #citiTon[5].Q )
      Coil( "Unit1.ControlNodes".citiMap.PMC.Machining_Assembly.Cycle_Time_Ready )
   END_RUNG
   RUNG wire#powerrail
      Contact( "Unit1.ControlNodes".citiMap.PMC.Machining_Assembly.Cycle_Time_Ready )
   END_RUNG wire#w1
   RUNG wire#powerrail
      Contact( "Unit1.ControlNodes".citiMap.PMC.Machining_Assembly.Cycle_Time_Ready )
      { S7_Templates := "time_type := Time" } #citiTon[5].TON(pt := #citi, et =>)
   END_RUNG
   // the same network as SCL:
   #_w1 := NOT (NOT "Unit1.ControlNodes".citiMap.PMC.Machining_Assembly.IncrGood_Count AND NOT "Unit1.ControlNodes".citiMap.PMC.Machining_Assembly.IncrReject_Count);
   #_w2 := #_w1 AND NOT #citi_Ptrig[5];   // rising edge
   #citi_Ptrig[5] := #_w1;
   "Unit1.ControlNodes".citiMap.PMC.Machining_Assembly.Cycle_Time_Ready := (#_w2 OR "Unit1.ControlNodes".citiMap.PMC.Machining_Assembly.Cycle_Time_Ready) AND NOT #citiTon[5].Q;
   #citiTon[5].TON(IN := "Unit1.ControlNodes".citiMap.PMC.Machining_Assembly.Cycle_Time_Ready, PT := #citi);
END_REGION

REGION Network 135: Fault bit Level1 6
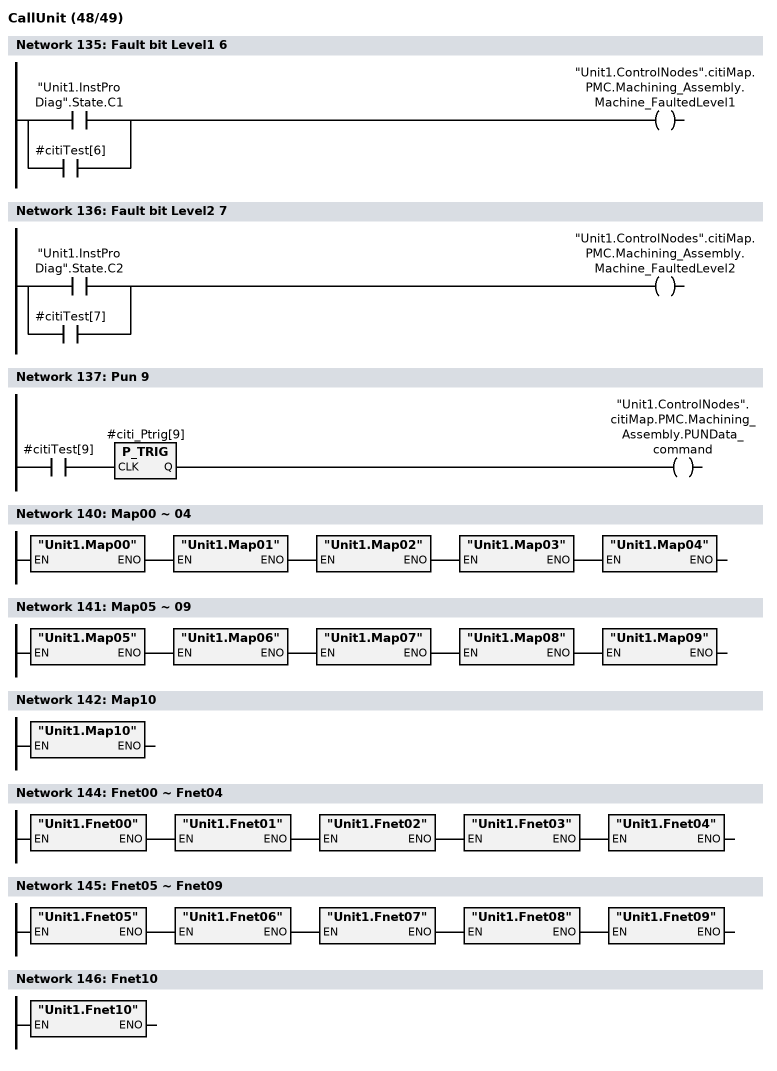
   RUNG wire#powerrail
      Contact( "Unit1.InstProDiag".State.C1 )
      wire#w1
      Coil( "Unit1.ControlNodes".citiMap.PMC.Machining_Assembly.Machine_FaultedLevel1 )
   END_RUNG
   RUNG wire#powerrail
      Contact( #citiTest[6] )
   END_RUNG wire#w1
   // the same network as SCL:
   "Unit1.ControlNodes".citiMap.PMC.Machining_Assembly.Machine_FaultedLevel1 := "Unit1.InstProDiag".State.C1 OR #citiTest[6];
END_REGION

REGION Network 136: Fault bit Level2 7
   RUNG wire#powerrail
      Contact( "Unit1.InstProDiag".State.C2 )
      wire#w1
      Coil( "Unit1.ControlNodes".citiMap.PMC.Machining_Assembly.Machine_FaultedLevel2 )
   END_RUNG
   RUNG wire#powerrail
      Contact( #citiTest[7] )
   END_RUNG wire#w1
   // the same network as SCL:
   "Unit1.ControlNodes".citiMap.PMC.Machining_Assembly.Machine_FaultedLevel2 := "Unit1.InstProDiag".State.C2 OR #citiTest[7];
END_REGION

REGION Network 137: Pun 9
   RUNG wire#powerrail
      Contact( #citiTest[9] )
      P_Trig( #citi_Ptrig[9] )
      Coil( "Unit1.ControlNodes".citiMap.PMC.Machining_Assembly.PUNData_command )
   END_RUNG
   // the same network as SCL:
   #_w1 := #citiTest[9] AND NOT #citi_Ptrig[9];   // rising edge
   #citi_Ptrig[9] := #citiTest[9];
   "Unit1.ControlNodes".citiMap.PMC.Machining_Assembly.PUNData_command := #_w1;
END_REGION

REGION Network 138: ControlNodes.CitiMap -> Unit1. EmNodes.Andon X
END_REGION

REGION Network 140: Map00 ~ 04
   RUNG wire#powerrail
      "Unit1.Map00"()
      "Unit1.Map01"()
      "Unit1.Map02"()
      "Unit1.Map03"()
      "Unit1.Map04"()
   END_RUNG
   // the same network as SCL:
   "Unit1.Map00"(ENO => #_w1);
   "Unit1.Map01"(EN := #_w1, ENO => #_w2);
   "Unit1.Map02"(EN := #_w2, ENO => #_w3);
   "Unit1.Map03"(EN := #_w3, ENO => #_w4);
   IF #_w4 THEN "Unit1.Map04"(); END_IF;
END_REGION

REGION Network 141: Map05 ~ 09
   RUNG wire#powerrail
      "Unit1.Map05"()
      "Unit1.Map06"()
      "Unit1.Map07"()
      "Unit1.Map08"()
      "Unit1.Map09"()
   END_RUNG
   // the same network as SCL:
   "Unit1.Map05"(ENO => #_w1);
   "Unit1.Map06"(EN := #_w1, ENO => #_w2);
   "Unit1.Map07"(EN := #_w2, ENO => #_w3);
   "Unit1.Map08"(EN := #_w3, ENO => #_w4);
   IF #_w4 THEN "Unit1.Map09"(); END_IF;
END_REGION

REGION Network 142: Map10
   RUNG wire#powerrail
      "Unit1.Map10"()
   END_RUNG
   // the same network as SCL:
   "Unit1.Map10"();
END_REGION

REGION Network 144: Fnet00 ~ Fnet04
   RUNG wire#powerrail
      "Unit1.Fnet00"()
      "Unit1.Fnet01"()
      "Unit1.Fnet02"()
      "Unit1.Fnet03"()
      "Unit1.Fnet04"()
   END_RUNG
   // the same network as SCL:
   "Unit1.Fnet00"(ENO => #_w1);
   "Unit1.Fnet01"(EN := #_w1, ENO => #_w2);
   "Unit1.Fnet02"(EN := #_w2, ENO => #_w3);
   "Unit1.Fnet03"(EN := #_w3, ENO => #_w4);
   IF #_w4 THEN "Unit1.Fnet04"(); END_IF;
END_REGION

REGION Network 145: Fnet05 ~ Fnet09
   RUNG wire#powerrail
      "Unit1.Fnet05"()
      "Unit1.Fnet06"()
      "Unit1.Fnet07"()
      "Unit1.Fnet08"()
      "Unit1.Fnet09"()
   END_RUNG
   // the same network as SCL:
   "Unit1.Fnet05"(ENO => #_w1);
   "Unit1.Fnet06"(EN := #_w1, ENO => #_w2);
   "Unit1.Fnet07"(EN := #_w2, ENO => #_w3);
   "Unit1.Fnet08"(EN := #_w3, ENO => #_w4);
   IF #_w4 THEN "Unit1.Fnet09"(); END_IF;
END_REGION

REGION Network 146: Fnet10
   RUNG wire#powerrail
      "Unit1.Fnet10"()
   END_RUNG
   // the same network as SCL:
   "Unit1.Fnet10"();
END_REGION

REGION Network 147: ******************** Q-DAS(=V-Gage) ********************
END_REGION

REGION Network 148: Call LMQTT_Client
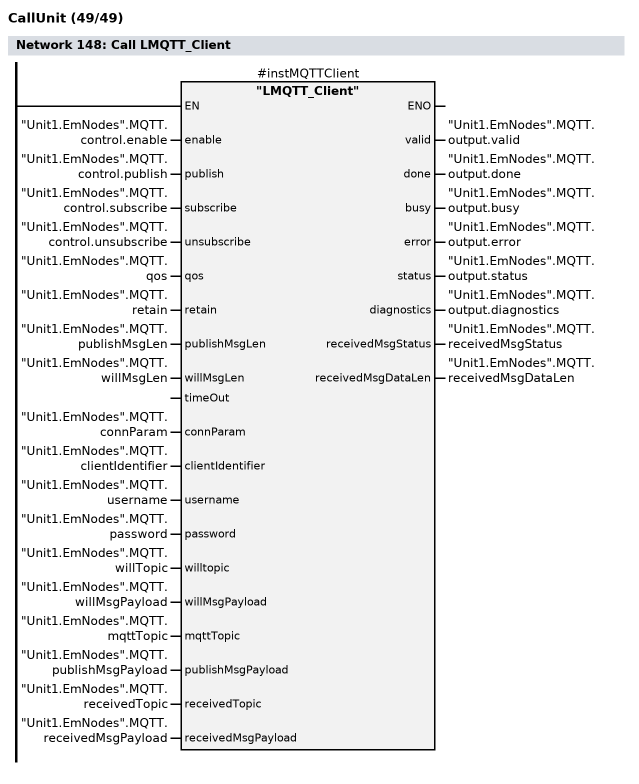
   RUNG wire#powerrail
      #instMQTTClient(enable := "Unit1.EmNodes".MQTT.control.enable, publish := "Unit1.EmNodes".MQTT.control.publish, subscribe := "Unit1.EmNodes".MQTT.control.subscribe, unsubscribe := "Unit1.EmNodes".MQTT.control.unsubscribe, qos := "Unit1.EmNodes".MQTT.qos, retain := "Unit1.EmNodes".MQTT.retain, publishMsgLen := "Unit1.EmNodes".MQTT.publishMsgLen, willMsgLen := "Unit1.EmNodes".MQTT.willMsgLen, timeOut :=, connParam := "Unit1.EmNodes".MQTT.connParam, clientIdentifier := "Unit1.EmNodes".MQTT.clientIdentifier, username := "Unit1.EmNodes".MQTT.username, password := "Unit1.EmNodes".MQTT.password, willtopic := "Unit1.EmNodes".MQTT.willTopic, willMsgPayload := "Unit1.EmNodes".MQTT.willMsgPayload, mqttTopic := "Unit1.EmNodes".MQTT.mqttTopic, publishMsgPayload := "Unit1.EmNodes".MQTT.publishMsgPayload, receivedTopic := "Unit1.EmNodes".MQTT.receivedTopic, receivedMsgPayload := "Unit1.EmNodes".MQTT.receivedMsgPayload, valid => "Unit1.EmNodes".MQTT.output.valid, done => "Unit1.EmNodes".MQTT.output.done, busy => "Unit1.EmNodes".MQTT.output.busy, error => "Unit1.EmNodes".MQTT.output.error, status => "Unit1.EmNodes".MQTT.output.status, diagnostics => "Unit1.EmNodes".MQTT.output.diagnostics, receivedMsgStatus => "Unit1.EmNodes".MQTT.receivedMsgStatus, receivedMsgDataLen => "Unit1.EmNodes".MQTT.receivedMsgDataLen)
   END_RUNG
   // the same network as SCL:
   #instMQTTClient(enable := "Unit1.EmNodes".MQTT.control.enable,   // "LMQTT_Client"
                   publish := "Unit1.EmNodes".MQTT.control.publish,
                   subscribe := "Unit1.EmNodes".MQTT.control.subscribe,
                   unsubscribe := "Unit1.EmNodes".MQTT.control.unsubscribe,
                   qos := "Unit1.EmNodes".MQTT.qos,
                   retain := "Unit1.EmNodes".MQTT.retain,
                   publishMsgLen := "Unit1.EmNodes".MQTT.publishMsgLen,
                   willMsgLen := "Unit1.EmNodes".MQTT.willMsgLen,
                   connParam := "Unit1.EmNodes".MQTT.connParam,
                   clientIdentifier := "Unit1.EmNodes".MQTT.clientIdentifier,
                   username := "Unit1.EmNodes".MQTT.username,
                   password := "Unit1.EmNodes".MQTT.password,
                   willtopic := "Unit1.EmNodes".MQTT.willTopic,
                   willMsgPayload := "Unit1.EmNodes".MQTT.willMsgPayload,
                   mqttTopic := "Unit1.EmNodes".MQTT.mqttTopic,
                   publishMsgPayload := "Unit1.EmNodes".MQTT.publishMsgPayload,
                   receivedTopic := "Unit1.EmNodes".MQTT.receivedTopic,
                   receivedMsgPayload := "Unit1.EmNodes".MQTT.receivedMsgPayload,
                   valid => "Unit1.EmNodes".MQTT.output.valid,
                   done => "Unit1.EmNodes".MQTT.output.done,
                   busy => "Unit1.EmNodes".MQTT.output.busy,
                   error => "Unit1.EmNodes".MQTT.output.error,
                   status => "Unit1.EmNodes".MQTT.output.status,
                   diagnostics => "Unit1.EmNodes".MQTT.output.diagnostics,
                   receivedMsgStatus => "Unit1.EmNodes".MQTT.receivedMsgStatus,
                   receivedMsgDataLen => "Unit1.EmNodes".MQTT.receivedMsgDataLen);
END_REGION

REGION Network 149: ******************** QR Handy Reader [Currently Unused] ********************
END_REGION
END_FUNCTION_BLOCK
